FUNCTION_BLOCK "GCS7_LiftingDevice"	// FB 85
TITLE = MACHINE: Lifting Device
//  
//COPYRIGHT:    (C) 1997  BUHLER AG, CH-9240 UZWIL,  SWITZERLAND
//
//PRODUCT:      GCS7
//
//TITLE:        FB 85 MACHINE: Lifting Device (de:Hubzug)
// 
//-------------------------------------------------------------------------
//
//IDENT:        AUTHOR:             DEPT:                       DATE:
//FB85.2.4      M.Wedler            AEB31                       28-Jul-2008
//              Software counter with functions hardware's counter
//FB85.2.3      U.Kemmesies         AEB31                       07-Dez-2007
//              No Counter-Card
//FB85.2.2      M.Wedler            AEB31                       05-Jan-2007
//              BankingLoadingScrew for kilning box, calibration,
//              load counter value after failure, InEnableLowerMinPos
//FB85.2.1      M.Wedler            AEB31                       12-Sep-2006
//              Don't initialisation way counter by loading counter value
//FB85.2.0      A.Egli              CT3                         22-Mar-2006
//              ParPulseOnTime,ParPulseOffTime
//FB85.1.0      A.Egli              CT3                         22-Mar-2006
//              1st Release in S7
//
//-------------------------------------------------------------------------
//
//PURPOSE:      MANUAL : see [LL.xxMAN]
//
//RESTRICTIONS: S7
//
//-------------------------------------------------------------------------
//
AUTHOR : EA
FAMILY : GCS7LL
NAME : Lifting
VERSION : 2.3
VAR
  Ma : UDT 20850;
  MotorLeft : FB 12;	//Element Motor
  MotorRight : FB 12;	//Element Motor
  LSTopLeft : FB 14;	//LS top left side
  LSTopRight : FB 14;	//LS top right side
  LSTopStopLeft : FB 14;	//Emergency stop stop left
  LSTopStopRight : FB 14;	//Emergency stop stop right
  SMLeft : FB 14;	//Speed monitoring left side
  SMRight : FB 14;	//Speed monitoring right side
  OffTrackMon : FB 14;	//Track monitoring
  CounterLeft : UDT 20851;
  CounterRight : UDT 20851;
END_VAR
VAR_TEMP
  tmpFaultSum : BOOL ;
  tmpEnable : BOOL ;
  tmpLocal : BOOL ;
  tmpLenDyn : INT ;
  tmpOK : BOOL ;
  tmpDiff : INT ;
  tmpAddrIOLeft : DINT ;
  tmpAddrIORight : DINT ;
  tmpAddrCounterLeft : DINT ;
  tmpAddrCounterRight : DINT ;
  tmpAddrOffset : DINT ;
  tmpUnloadingActive : BOOL ;
END_VAR
BEGIN
NETWORK
TITLE =
      L     90;
      T     #tmpLenDyn;
NETWORK
TITLE = PC Control
//=== Test Object number =====================
      L     "SYS_DirectCtrlDB".PC.ObjectNo;	//PCControl.ObjectNo
      L     #Ma.Par.ParObjectNo;	//Input ObjectNo
      <>I;
      JC    aEnd;
//=== Test OType      ========================
      L     2085;	//Input object type
      L     "SYS_DirectCtrlDB".PC.ObjectType;	//PCControl.ObjectType
      <>I;
      JC    aEnd;
//=== Test Handshake =========================
      A     "SYS_DirectCtrlDB".PC.Hsk.FExamine;	// Handshake.FExamine
      JC    aExa;
      A     "SYS_DirectCtrlDB".PC.Hsk.FDefineCmd;	// Handshake.FDefineCmd
      O     "SYS_DirectCtrlDB".PC.Hsk.FDefinePara;	// Handshake.FDefinePara
      JC    aCmd;
      JU    aEnd;
// Write new commands from PC to Interface of group 
aCmd: A     "SYS_DirectCtrlDB".PC.Cmd1[8];	//Cmd1[8]=CmdOff
      S     #Ma.CmdOff;
      A     "SYS_DirectCtrlDB".PC.Cmd1[9];	//Cmd1[9]=CmdUp
      S     #Ma.CmdUp;
      A     "SYS_DirectCtrlDB".PC.Cmd1[10];	//Cmd1[10]=CmdNext
      S     #Ma.CmdNext;
      A     "SYS_DirectCtrlDB".PC.Cmd1[11];	//Cmd1[11]=CmdFaultReset
      S     #Ma.CmdFaultReset;
      A     "SYS_DirectCtrlDB".PC.Cmd1[13];	//Cmd1[13]=CmdManualOn
      S     #Ma.InManual;
      A     "SYS_DirectCtrlDB".PC.Cmd1[7];	//Cmd1[6]=CmdDown
      S     #Ma.CmdDown;
      A     "SYS_DirectCtrlDB".PC.Cmd2[13];	//Cmd2[13]=CmdManualOff
      R     #Ma.InManual;
//-----------------------------------------------------------
//Audit Log
aExa: NOP   0;
//------------------------------------------
      TAR2;	// Address Dynamic datas
      T     "SYS_DirectCtrlDB".GC.InDynAddr;	// -->PCControl.GC.InDynAddr
      L     #tmpLenDyn;	// Length Dynamic data
      T     "SYS_DirectCtrlDB".GC.InDynLen;	// -->PCControl.GC.InDynLen
      L     0;
      T     "SYS_DirectCtrlDB".GC.InParaAddr;	// -->PCControl.GC.InParaAddr
      T     "SYS_DirectCtrlDB".GC.InParaLen;	// -->PCControl.GC.InParaLen
      L     1;	// Code FcExamine
      UC    "SYS_DirectCtrl";
      L     10;	//Revision
      T     "SYS_DirectCtrlDB".GC.Revision;
aEnd: NOP   0;
NETWORK
TITLE = Calculate Address for Counter
      NOP   0;
//Calculate address for counter
      TAR2;
      L     DW#16#FFFFFF;
      AD;
      T     #tmpAddrOffset;
      L     P##CounterLeft;
      +D;
      T     #tmpAddrCounterLeft;
      L     #Ma.Par.ParIOByteNoCounterLeft;
      SLD   3;
      T     #tmpAddrIOLeft;
      L     #tmpAddrOffset;
      L     P##CounterRight;
      +D;
      T     #tmpAddrCounterRight;
      L     #Ma.Par.ParIOByteNoCounterRight;
      SLD   3;
      T     #tmpAddrIORight;
NETWORK
TITLE = Commands for Counter
//      L     0                           // [2.3]
//      L     #tmpAddrIOLeft              // [2.3]
//      ==D                               // [2.3]
////[2.4]     SPB   CTX0                        // [2.3]
//      SPB   IUK1                        // [2.4]
//      SPA   IUK0                        // [2.4]
//IUK1: NOP   0                           // [2.4]
////Calibration Zero                      // [2.4]
//      U     #Ma.InCalibration           // [2.4]
//      U     #Ma.InCalibrationZero       // [2.4]
//      U     #Ma.InPowerOk               // [2.4]
//      U     #Ma.InPowerOkDelayDone      // [2.4]
//      SPBN  IUK2                        // [2.4]
//      L     L#0                         // [2.4]
//      T     #CounterLeft.OutpSetCount   // [2.4]
//      T     #CounterRight.OutpSetCount  // [2.4]
//      T     #CounterLeft.VarInpHold     // [2.4]
//      T     #CounterRight.VarInpHold    // [2.4]
//      SET                               // [2.4]
//      S     #CounterLeft.OutpLOAD_VAL   // [2.4]
//      S     #CounterRight.OutpLOAD_VAL  // [2.4]
//IUK2: NOP   0                           // [2.4]
//      U     #CounterLeft.InpSTS_LOAD    // [2.4]
//      R     #CounterLeft.OutpLOAD_VAL   // [2.4]
//      U     #CounterRight.InpSTS_LOAD   // [2.4]
//      R     #CounterRight.OutpLOAD_VAL  // [2.4]
//      SPA   CTX0                        // [2.4]
//IUK0: NOP   0
      L     0;	// [2.3]
      L     #tmpAddrIOLeft;	// [2.3]
      ==D;	// [2.3]
//[2.4]     SPB   CTX0                        // [2.3]
      JC    IUK1;	// [2.4]
      JU    IUK0;	// [2.4]
IUK1: NOP   0;	// [2.4]
//Calibration Zero                      // [2.4]
      A     #Ma.InCalibration;	// [2.4]
      A     #Ma.InCalibrationZero;	// [2.4]
      A     #Ma.InPowerOk;	// [2.4]
      A     #Ma.InPowerOkDelayDone;	// [2.4]
      JCN   IUK2;	// [2.4]
      L     L#0;	// [2.4]
      T     #CounterLeft.InpActCount;	// [2.4]
      T     #CounterRight.InpActCount;	// [2.4]
      T     #CounterLeft.VarInpHold;	// [2.4]
      T     #CounterRight.VarInpHold;	// [2.4]
IUK2: NOP   0;	// [2.4]
      JU    CTX0;	// [2.4]
IUK0: NOP   0;
      NOP   0;
//Clear command or counter
      A     #Ma.InPowerOk;	// [2.2]
      A     #CounterLeft.OutpLOAD_VAL;	// [2.2]
      AN    #CounterLeft.InpSTS_LOAD;	// [2.2]
      JC    CTJ9;	// [2.2]
      LAR1  #tmpAddrCounterLeft;
      L     0;
      T     DID [AR1,P#4.0];
CTJ9: NOP   0;	// [2.2]
      A     #Ma.InPowerOk;	// [2.2]
      A     #CounterRight.OutpLOAD_VAL;	// [2.2]
      AN    #CounterRight.InpSTS_LOAD;	// [2.2]
      JC    CTJ8;	// [2.2]
      LAR1  #tmpAddrCounterRight;
      L     0;
      T     DID [AR1,P#4.0];
CTJ8: NOP   0;	// [2.2]
//---------------------------
      SET;
      S     #CounterLeft.OutpSW_GATE;
      S     #CounterRight.OutpSW_GATE;
//---------------------------
//Load counter value after failure      // [2.2]
      A     #Ma.InPowerOk;
      AN    #Ma.InPowerOkDelayDone;
      O;	// [2.2]
      A     #CounterLeft.OutpLOAD_VAL;	// [2.2]
      AN    #CounterLeft.InpSTS_LOAD;	// [2.2]
      JCN   CTJ2;	// [2.2]
      L     #CounterLeft.VarInpHold;
      T     #CounterLeft.OutpSetCount;
//    SET                               // [2.2]
      L     #CounterLeft.VarInpHold;	// [2.2]
      L     #CounterLeft.InpActCount;	// [2.2]
      <>D;	// [2.2]
      S     #CounterLeft.OutpLOAD_VAL;
CTJ2: NOP   0;	// [2.2]
      A     #Ma.InPowerOk;
      AN    #Ma.InPowerOkDelayDone;
      O;	// [2.2]
      A     #CounterRight.OutpLOAD_VAL;	// [2.2]
      AN    #CounterRight.InpSTS_LOAD;	// [2.2]
      JCN   CTJ1;
      L     #CounterRight.VarInpHold;
      T     #CounterRight.OutpSetCount;
//    SET                               // [2.2]
      L     #CounterRight.VarInpHold;	// [2.2]
      L     #CounterRight.InpActCount;	// [2.2]
      <>D;	// [2.2]
      S     #CounterRight.OutpLOAD_VAL;
CTJ1: NOP   0;
      A     #Ma.InPowerOk;
      A     #Ma.InPowerOkDelayDone;
      AN    #CounterLeft.InpSTS_LOAD;	// [2.2]
      AN    #CounterRight.InpSTS_LOAD;	// [2.2]
      AN    #CounterLeft.OutpLOAD_VAL;	// [2.2]
      AN    #CounterRight.OutpLOAD_VAL;	// [2.2]
      JCN   CTJ0;
      L     #CounterLeft.InpActCount;
      T     #CounterLeft.VarInpHold;
      L     #CounterRight.InpActCount;
      T     #CounterRight.VarInpHold;
CTJ0: NOP   0;
//Calibration Zero                      // [2.2]
      A     #Ma.InCalibration;	// [2.2]
      A     #Ma.InCalibrationZero;	// [2.2]
      A     #Ma.InPowerOk;	// [2.2]
      A     #Ma.InPowerOkDelayDone;	// [2.2]
      JCN   CTZ0;	// [2.2]
      L     L#0;	// [2.2]
      T     #CounterLeft.OutpSetCount;	// [2.2]
      T     #CounterRight.OutpSetCount;	// [2.2]
      T     #CounterLeft.VarInpHold;	// [2.2]
      T     #CounterRight.VarInpHold;	// [2.2]
      SET;	// [2.2]
      S     #CounterLeft.OutpLOAD_VAL;	// [2.2]
      S     #CounterRight.OutpLOAD_VAL;	// [2.2]
CTZ0: NOP   0;	// [2.2]
      A     #CounterLeft.InpSTS_LOAD;	// [2.2]
      R     #CounterLeft.OutpLOAD_VAL;	// [2.2]
      A     #CounterRight.InpSTS_LOAD;	// [2.2]
      R     #CounterRight.OutpLOAD_VAL;	// [2.2]
CTX0: NOP   0;	// [2.3]
NETWORK
TITLE = Initialisation way counter when in upper finally position 
//      L     0                           // [2.3]
//      L     #tmpAddrIOLeft              // [2.3]
//      ==D                               // [2.3]
////[2.4]      SPB   M050                        // [2.3]
//      SPB   UKI1                        // [2.4]
//      SPA   UKI0                        // [2.4]
//UKI1: NOP   0                           // [2.4]
//      UN    #Ma.InPowerOkDelayDone      // [2.4]
//      O     #Ma.InCalibration           // [2.4]
//      SPB   UKI2                        // [2.4]
//// Initialisation counter left when in end position top
//      O     #MotorLeft.StStartedFwd
//      O     #MotorLeft.StStopping
//      U     #LSTopLeft.StTrue
//      SPBN  UKI2
//      L     #Ma.Par.ParPositionTopLeftInc
//      ITD   
//      T     #CounterLeft.OutpSetCount
//      T     #CounterLeft.VarInpHold     // [2.4]
//      SET                               // [2.4]
//      S     #CounterLeft.OutpLOAD_VAL   // [2.4]
//UKI2: NOP   0
//      UN    #Ma.InPowerOkDelayDone      // [2.4]
//      O     #Ma.InCalibration           // [2.4]
//      SPB   UKI3                        // [2.4]
//// Initialisation counter rigth  when in end position top
//      O     #MotorRight.StStartedFwd
//      O     #MotorRight.StStopping
//      U     #LSTopRight.StTrue          // Endschalter oben
//      SPBN  UKI3
//      L     #Ma.Par.ParPositionTopRightInc
//      ITD   
//      T     #CounterRight.OutpSetCount
//      T     #CounterRight.VarInpHold    // [2.4]
//      SET                               // [2.4]
//      S     #CounterRight.OutpLOAD_VAL  // [2.4]
//UKI3: NOP   0                           // [2.4]
//      U     #CounterLeft.InpSTS_LOAD    // [2.4]
//      R     #CounterLeft.OutpLOAD_VAL   // [2.4]
//      U     #CounterRight.InpSTS_LOAD   // [2.4]
//      R     #CounterRight.OutpLOAD_VAL  // [2.4]
//      SPA   M050                        // [2.4]
//UKI0: NOP   0                           // [2.4]
//
      L     0;	// [2.3]
      L     #tmpAddrIOLeft;	// [2.3]
      ==D;	// [2.3]
//[2.4]      SPB   M050                        // [2.3]
      JC    UKI1;	// [2.4]
      JU    UKI0;	// [2.4]
UKI1: NOP   0;	// [2.4]
      AN    #Ma.InPowerOkDelayDone;	// [2.4]
      O     #Ma.InCalibration;	// [2.4]
      JC    UKI2;	// [2.4]
// Initialisation counter left when in end position top
      O     #MotorLeft.StStartedFwd;
      O     #MotorLeft.StStopping;
      A     #LSTopLeft.StTrue;
      JCN   UKI2;
      L     #Ma.Par.ParPositionTopLeftInc;
      ITD;
      T     #CounterLeft.InpActCount;	// [2.4]
      T     #CounterLeft.VarInpHold;	// [2.4]
UKI2: NOP   0;
      AN    #Ma.InPowerOkDelayDone;	// [2.4]
      O     #Ma.InCalibration;	// [2.4]
      JC    UKI3;	// [2.4]
// Initialisation counter rigth  when in end position top
      O     #MotorRight.StStartedFwd;
      O     #MotorRight.StStopping;
      A     #LSTopRight.StTrue;	// Endschalter oben
      JCN   UKI3;
      L     #Ma.Par.ParPositionTopRightInc;
      ITD;
      T     #CounterRight.InpActCount;	// [2.4]
      T     #CounterRight.VarInpHold;	// [2.4]
UKI3: NOP   0;	// [2.4]
      JU    M050;	// [2.4]
UKI0: NOP   0;	// [2.4]
      NOP   0;
//-------------------------------------------------------
      A     #CounterLeft.InpSTS_LOAD;	// [2.1]
      ON    #Ma.InPowerOkDelayDone;	// [2.1]
      O     #Ma.InCalibration;	// [2.2]
      JC    M051;	// [2.1]
// Initialisation counter left when in end position top
      O     #MotorLeft.StStartedFwd;
      O     #MotorLeft.StStopping;
      A     #LSTopLeft.StTrue;
      JCN   M051;
      L     #Ma.Par.ParPositionTopLeftInc;
      ITD;
      T     #CounterLeft.OutpSetCount;
      T     #CounterLeft.VarInpHold;	// [2.2]
//Set Write command 
      L     #Ma.Par.ParPositionTopLeftInc;
      L     #Ma.OutIncrementLeft;
      <>I;
      S     #CounterLeft.OutpLOAD_VAL;	//--> Command to counter to set target value
M051: NOP   0;
//-------------------------------------------------------
      A     #CounterRight.InpSTS_LOAD;	// [2.1]
      ON    #Ma.InPowerOkDelayDone;	// [2.1]
      O     #Ma.InCalibration;	// [2.2]
      JC    M052;	// [2.1]
// Initialisation counter rigth  when in end position top
      O     #MotorRight.StStartedFwd;
      O     #MotorRight.StStopping;
      A     #LSTopRight.StTrue;	// Endschalter oben
      JCN   M052;
      L     #Ma.Par.ParPositionTopRightInc;
      ITD;
      T     #CounterRight.OutpSetCount;
      T     #CounterRight.VarInpHold;	// [2.2]
//Set Write command
      L     #Ma.Par.ParPositionTopRightInc;
      L     #Ma.OutIncrementRight;
      <>I;
      S     #CounterRight.OutpLOAD_VAL;	//--> Command to counter to set target value
M052: NOP   0;
M050: NOP   0;	// [2.3]
NETWORK
TITLE = Read Global Command
      A     "GCS7_Gr_OutFaultReset";	// OutFaultReset
      S     #Ma.CmdFaultReset;
NETWORK
TITLE = Write Outputs of counter
      L     0;
      L     #tmpAddrIOLeft;
      ==D;
      JC    WCJ0;
//Write Outputs  Counter left
      LAR1  #tmpAddrCounterLeft;
      L     DID [AR1,P#0.0];
      LAR1  #tmpAddrIOLeft;
      T     PQD [AR1,P#0.0];
      LAR1  #tmpAddrCounterLeft;
      L     DID [AR1,P#4.0];
      LAR1  #tmpAddrIOLeft;
      T     PQD [AR1,P#4.0];
//Write Outputs Counter right
      LAR1  #tmpAddrCounterRight;
      L     DID [AR1,P#0.0];
      LAR1  #tmpAddrIORight;
      T     PQD [AR1,P#0.0];
      LAR1  #tmpAddrCounterRight;
      L     DID [AR1,P#4.0];
      LAR1  #tmpAddrIORight;
      T     PQD [AR1,P#4.0];
WCJ0: NOP   0;
NETWORK
TITLE = Read Counter
      L     0;
      L     #tmpAddrIOLeft;
      ==D;
      JC    WRJ0;
//Read IO Counter left
      LAR1  #tmpAddrIOLeft;
      L     PID [AR1,P#0.0];
      LAR1  #tmpAddrCounterLeft;
      T     DID [AR1,P#8.0];
      LAR1  #tmpAddrIOLeft;
      L     PID [AR1,P#4.0];
      LAR1  #tmpAddrCounterLeft;
      T     DID [AR1,P#12.0];
//Read IO Counter right
      LAR1  #tmpAddrIORight;
      L     PID [AR1,P#0.0];
      LAR1  #tmpAddrCounterRight;
      T     DID [AR1,P#8.0];
      LAR1  #tmpAddrIORight;
      L     PID [AR1,P#4.0];
      LAR1  #tmpAddrCounterRight;
      T     DID [AR1,P#12.0];
WRJ0: NOP   0;
NETWORK
TITLE = Calculate: mm per incement 
      L     #Ma.Par.ParPositionTopLeftUnits;
      DTR;
      L     #Ma.Par.ParPositionTopLeftInc;	//Hoehe Endschalter 
      DTR;
      /R;
      T     #Ma.Par.OutUnitsPerIncLeft;
      L     #Ma.Par.ParPositionTopRightUnits;
      DTR;
      L     #Ma.Par.ParPositionTopRightInc;	//Hoehe Endschalter 
      DTR;
      /R;
      T     #Ma.Par.OutUnitsPerIncRight;
NETWORK
TITLE = Speed Monitoring Lifting 
      NOP   0;
//==========================================================
//Speed Monitoring Left
//==========================================================
//- Check if increment is changing
      A(;
      L     #CounterLeft.InpActCount;
      L     #Ma.OutIncrementLeft;
      ==D;
      );
      A(;
      O     #MotorLeft.OutpRunFwd;
      O     #MotorLeft.OutpRunRev;
      );
      AN    #Ma.CmdFaultReset;
      JC    M1J1;
      L     #Ma.Par.ParMonTime;	//5s
      T     #Ma.Par.OutMonTimeLeft;
      S     #SMLeft.InpTrue;
//---Run monitoring time
M1J1: AN    "GCS7_Gr_OutTick200ms";
      JC    M1J2;
      L     #Ma.Par.OutMonTimeLeft;
      +     -2;
      T     #Ma.Par.OutMonTimeLeft;
      L     0;
      >=I;
      JC    M1J2;
      T     #Ma.Par.OutMonTimeLeft;
      R     #SMLeft.InpTrue;
//---Store old counter value
M1J2: L     #CounterLeft.InpActCount;
      T     #Ma.OutIncrementLeft;
//==========================================================
//Speed Monitoring Right
//==========================================================
//- Check if increment is changing
      A(;
      L     #CounterRight.InpActCount;
      L     #Ma.OutIncrementRight;
      ==D;
      );
      A(;
      O     #MotorRight.OutpRunFwd;
      O     #MotorRight.OutpRunRev;
      );
      AN    #Ma.CmdFaultReset;
      JC    M2J1;
      L     #Ma.Par.ParMonTime;	//5s
      T     #Ma.Par.OutMonTimeRight;
      S     #SMRight.InpTrue;
//---Run monitoring time
M2J1: AN    "GCS7_Gr_OutTick200ms";
      JC    M2J2;
      L     #Ma.Par.OutMonTimeRight;
      +     -2;
      T     #Ma.Par.OutMonTimeRight;
      L     0;
      >=I;
      JC    M2J2;
      T     #Ma.Par.OutMonTimeRight;
      R     #SMRight.InpTrue;
//---Store old counter value
M2J2: L     #CounterRight.InpActCount;
      T     #Ma.OutIncrementRight;
NETWORK
TITLE = Calculation position in mm
// Zaehlwert Hubzug 1 in mm umrechnen
      L     #Ma.OutIncrementLeft;
      DTR;
      L     #Ma.Par.OutUnitsPerIncLeft;
      *R;
      RND;
      T     #Ma.OutPositionLeft;
// Zaehlwert Hubzug 2 in mm umrechnen
      L     #Ma.OutIncrementRight;
      DTR;
      L     #Ma.Par.OutUnitsPerIncRight;
      *R;
      RND;
      T     #Ma.OutPositionRight;
NETWORK
TITLE = Check maximum difference position to stop 1 motor 
      NOP   0;
//---Check Position left to high
      L     #Ma.OutPositionLeft;
      L     #Ma.BankingLoadingScrew;	// [2.2]
      +I;	// [2.2]
      L     #Ma.OutPositionRight;
      -I;
      T     #Ma.OutPositionDifference;
      L     #Ma.Par.ParMaxOffTrackPause;
      >=I;
      S     #Ma.OutPositionLeftToHigh;
      L     #Ma.OutPositionRight;
      L     #Ma.BankingLoadingScrew;	// [2.2]
      -I;	// [2.2]
      L     #Ma.OutPositionLeft;
      >=I;
      R     #Ma.OutPositionLeftToHigh;
//---Check position right to high
      L     #Ma.OutPositionRight;
      L     #Ma.BankingLoadingScrew;	// [2.2]
      -I;	// [2.2]
      L     #Ma.OutPositionLeft;
      -I;
      L     #Ma.Par.ParMaxOffTrackPause;
      >=I;
      S     #Ma.OutPositionRightToHigh;
      L     #Ma.OutPositionRight;
      L     #Ma.BankingLoadingScrew;	// [2.2]
      -I;	// [2.2]
      L     #Ma.OutPositionLeft;
      <=I;
      R     #Ma.OutPositionRightToHigh;
NETWORK
TITLE = Check maximum difference position to generate fault
      L     #Ma.OutPositionLeft;
      L     #Ma.OutPositionRight;
      -I;
      JP    DIJ1;
      NEGI;
DIJ1: L     #Ma.Par.ParMaxOffTrackFault;
      >=I;
      =     #Ma.OutDifferenceFault;
NETWORK
TITLE = Check Minimum position
      A(;
      L     #Ma.OutPositionLeft;
      L     #Ma.Par.ParPositionMin;
      >=I;
      );
      A(;
      L     #Ma.OutPositionRight;
      L     #Ma.Par.ParPositionMin;
      >=I;
      );
      =     #Ma.OutHigherMinPos;
NETWORK
TITLE = Check Adjusted
      NOP   0;
//------------------
      L     #Ma.OutPositionLeft;
      L     #Ma.InPositionTarget;
      -I;
      JP    A1J1;
      NEGI;
A1J1: L     #Ma.Par.ParTolPosition;
      <=I;
      =     #Ma.OutAdjustedLeft;
//------------------
      L     #Ma.OutPositionRight;
      L     #Ma.BankingLoadingScrew;	// [2.2]
      -I;	// [2.2]
      L     #Ma.InPositionTarget;
      -I;
      JP    A2J1;
      INVI;
A2J1: L     #Ma.Par.ParTolPosition;
      <=I;
      =     #Ma.OutAdjustedRight;
//------------------
NETWORK
TITLE = Interlocking
//===Global Group Orders===
      A     "GCS7_Gr_OutManualOff";	//Gr.OutManualOff
      R     #Ma.InManual;
      A     #Ma.InManual;
      S     "GCS7_Gr_InManual";	//Gr.InManual
//--------------
      A     #Ma.CmdUp;
      S     #Ma.OutManStartReqUp;
      R     #Ma.OutManStartReqDown;
      A     #Ma.CmdDown;
      R     #Ma.OutManStartReqUp;
      S     #Ma.OutManStartReqDown;
      A     #Ma.CmdOff;
      ON    #Ma.InManual;
      R     #Ma.OutManStartReqUp;
      R     #Ma.OutManStartReqDown;
//--- Fault----
      A     #MotorLeft.StFault;
      O     #MotorRight.StFault;
      O     #LSTopLeft.StFault;
      O     #LSTopRight.StFault;
      O     #LSTopStopLeft.StFault;
      O     #LSTopStopRight.StFault;
      O     #SMLeft.StFault;
      O     #SMRight.StFault;
      O     #OffTrackMon.StFault;
      =     #tmpFaultSum;
//--- InLocal----
      A     #Ma.InLocal;
      AN    #Ma.InManual;
      =     #tmpLocal;
      =     #MotorLeft.InLocal;
      =     #MotorRight.InLocal;
      =     #LSTopLeft.InLocal;
      =     #LSTopRight.InLocal;
      =     #LSTopStopLeft.InLocal;
      =     #LSTopStopRight.InLocal;
      =     #SMLeft.InLocal;
      =     #SMRight.InLocal;
      =     #OffTrackMon.InLocal;
//--- Fault Reset -------------
      A     #Ma.CmdFaultReset;
      S     #MotorLeft.CmdFaultReset;
      S     #MotorRight.CmdFaultReset;
      S     #LSTopLeft.CmdFaultReset;
      S     #LSTopRight.CmdFaultReset;
      S     #LSTopStopLeft.CmdFaultReset;
      S     #LSTopStopRight.CmdFaultReset;
      S     #SMLeft.CmdFaultReset;
      S     #SMRight.CmdFaultReset;
      S     #OffTrackMon.CmdFaultReset;
NETWORK
TITLE = Start as Pulse during unloading [2.0]
      A     #Ma.InEnableUp;	//[2.0]
      O     #Ma.InEnableDown;	//[2.0]
      AN    #tmpLocal;	//[2.0]
      AN    #Ma.InManual;	//[2.0]
      AN    #Ma.CmdOff;	//[2.0]
      AN    #Ma.StAdjusted;	//[2.0]
      AN    #tmpFaultSum;	//[2.0]
      A     #Ma.InUnloading;	//[2.0]
      =     #tmpUnloadingActive;	//[2.0]
      AN    #tmpUnloadingActive;	//[2.0]
      R     #Ma.OutPulseOn;	//[2.0]
      L     0;	//[2.0]
      JC    PuJ3;	//[2.0]
//--Decrement pulse time --
      AN    "GCS7_Gr_OutTick200ms";	//[2.0]
      L     #Ma.OutPulseTime;	//[2.0]
      JC    PuJ4;	//[2.0]
      +     -2;	//[2.0]
      T     #Ma.OutPulseTime;	//[2.0]
PuJ4: L     0;	//[2.0]
      >I;	//[2.0]
      JC    PuJ1;	//[2.0]
      AN    #Ma.OutPulseOn;	//[2.0]
      S     #Ma.OutPulseOn;	//[2.0]
      L     #Ma.Par.ParPulseOffTime;	//[2.0]
      JC    PuJ3;	//[2.0]
      R     #Ma.OutPulseOn;	//[2.0]
      L     #Ma.Par.ParPulseOnTime;	//[2.0]
PuJ3: T     #Ma.OutPulseTime;	//[2.0]
PuJ1: NOP   0;	//[2.0]
NETWORK
TITLE = Interlocking Motor Left
      L     #Ma.OutIncrementLeft;
      L     0;
      >I;
      AN    #tmpFaultSum;
      ON    #Ma.InInterlocked;
      A     #Ma.InEnableDown;
      A(;
      L     #Ma.InPositionTarget;
      L     #Ma.OutPositionLeft;
      <I;
      AN    #Ma.OutAdjustedLeft;
      AN    #Ma.InManual;
      A(;
      ON    #Ma.InUnloading;	//[2.0]
      ON    #Ma.OutPulseOn;	//[2.0]
      );
      O     #Ma.OutManStartReqDown;
      );
      AN    #Ma.OutPositionRightToHigh;
      AN    #Ma.OutDifferenceFault;
      A     #Ma.InEnableDown;
      A     #Ma.InEnableLowerMinPos;	//[2.2]
      A     #Ma.InPowerOkDelayDone;
      =     #MotorLeft.InEnableRev;
      AN    #tmpFaultSum;
      A     #LSTopLeft.StFalse;
      A     #LSTopStopLeft.StFalse;
      ON    #Ma.InInterlocked;
      A     #Ma.InEnableDown;
      A(;
      L     #Ma.InPositionTarget;
      L     #Ma.OutPositionLeft;
      >I;
      AN    #Ma.OutAdjustedLeft;
      AN    #Ma.InManual;
      A(;
      ON    #Ma.InUnloading;	//[2.0]
      ON    #Ma.OutPulseOn;	//[2.0]
      );
      O     #Ma.OutManStartReqUp;
      );
      AN    #Ma.OutPositionLeftToHigh;
      A     #Ma.InEnableUp;
      AN    #Ma.OutDifferenceFault;
      A     #Ma.InPowerOkDelayDone;
      =     #MotorLeft.InEnableFwd;
      A     #Ma.CmdNext;
      O     #Ma.InManual;
      S     #MotorLeft.CmdNext;
NETWORK
TITLE = Interlocking Motor Right
      L     #Ma.OutIncrementRight;
      L     0;
      >I;
      AN    #tmpFaultSum;
      ON    #Ma.InInterlocked;
      A     #Ma.InEnableDown;
      A(;
      L     #Ma.InPositionTarget;
      L     #Ma.BankingLoadingScrew;	//[2.2]
      +I;	//[2.2]
      L     #Ma.OutPositionRight;
      <I;
      AN    #Ma.OutAdjustedRight;
      AN    #Ma.InManual;
      A(;
      ON    #Ma.InUnloading;	//[2.0]
      ON    #Ma.OutPulseOn;	//[2.0]
      );
      O     #Ma.OutManStartReqDown;
      );
      AN    #Ma.OutPositionLeftToHigh;
      AN    #Ma.OutDifferenceFault;
      A     #Ma.InEnableDown;
      A     #Ma.InEnableLowerMinPos;	//[2.2]
      A     #Ma.InPowerOkDelayDone;
      =     #MotorRight.InEnableRev;
      AN    #tmpFaultSum;
      A     #LSTopRight.StFalse;
      A     #LSTopStopRight.StFalse;
      ON    #Ma.InInterlocked;
      A     #Ma.InEnableDown;
      A(;
      L     #Ma.InPositionTarget;
      L     #Ma.BankingLoadingScrew;	//[2.2]
      +I;	//[2.2]
      L     #Ma.OutPositionRight;
      >I;
      AN    #Ma.OutAdjustedRight;
      AN    #Ma.InManual;
      A(;
      ON    #Ma.InUnloading;	//[2.0]
      ON    #Ma.OutPulseOn;	//[2.0]
      );
      O     #Ma.OutManStartReqUp;
      );
      AN    #Ma.OutPositionRightToHigh;
      AN    #Ma.OutDifferenceFault;
      A     #Ma.InEnableUp;
      A     #Ma.InPowerOkDelayDone;
      =     #MotorRight.InEnableFwd;
      A     #Ma.CmdNext;
      O     #Ma.InManual;
      S     #MotorRight.CmdNext;
NETWORK
TITLE = Interlocking LSTopStopLeft, LSTopStopRight,LSTopLeft,LSTopRigh
//Mointoring false
//When started downwards, the the LS must be uncovered after 30 mm
//
//
      CLR;
      =     #LSTopStopLeft.InMonTrue;
      =     #LSTopStopRight.InMonTrue;
      CLR;
      =     #LSTopLeft.InMonTrue;
      =     #LSTopRight.InMonTrue;
//Monitoring false
      L     #Ma.Par.ParPositionTopLeftUnits;
      L     #Ma.OutPositionLeft;
      -I;
      L     30;	//30mms
      >=I;
      A     #MotorLeft.StStartedRev;
      A     #Ma.InInterlocked;
      =     #LSTopLeft.InMonFalse;
      SET;
      =     #LSTopStopLeft.InMonFalse;
      L     #Ma.Par.ParPositionTopRightUnits;
      L     #Ma.OutPositionRight;
      -I;
      L     30;	//30mms
      >=I;
      A     #MotorRight.StStartedRev;
      A     #Ma.InInterlocked;
      =     #LSTopRight.InMonFalse;
      SET;
      =     #LSTopStopRight.InMonFalse;
NETWORK
TITLE = Control Element SMLeft, SMRight
      A     #MotorLeft.StStartedRev;
      O     #MotorLeft.StStartedFwd;
      =     #SMLeft.InMonTrue;
      A     #MotorRight.StStartedRev;
      O     #MotorRight.StStartedFwd;
      =     #SMRight.InMonTrue;
NETWORK
TITLE = Control Element OffTrackMon
      AN    #Ma.OutDifferenceFault;
      =     #OffTrackMon.InpTrue;
      SET;
      =     #OffTrackMon.InMonTrue;
NETWORK
TITLE = Call Motor Left
      CALL  #MotorLeft;
NETWORK
TITLE = Call Motor Right
      CALL  #MotorRight;
NETWORK
TITLE = Call Digital Input: LSTopLeft
      CALL  #LSTopLeft;
NETWORK
TITLE = Call Digital Input: LSTopRight
      CALL  #LSTopRight;
NETWORK
TITLE = Call Digital Input: LSStopLeft
      CALL  #LSTopStopLeft;
NETWORK
TITLE = Call Digital Input: LSStopRight
      CALL  #LSTopStopRight;
NETWORK
TITLE = Call Digital Input: SMLeft
      CALL  #SMLeft;
NETWORK
TITLE = Call Digital Input: SMRight
      CALL  #SMRight;
NETWORK
TITLE = Call Digital Input: OffTrackMon
      CALL  #OffTrackMon;
NETWORK
TITLE = States
      A     #Ma.StStopped;
      JC    S0;
      A     #Ma.StAdjusted;
      JC    S6;
      A     #Ma.StStartedUP;
      JC    S2;
      A     #Ma.StStartedDown;
      JC    S5;
      A     #Ma.StStopping;
      JC    S3;
      A     #Ma.StStarting;
      JC    S1;
      A     #Ma.StFault;
      JC    S4;
      JU    xxS0;	//Initialise: goto StStopped
NETWORK
TITLE = StStopped
xxS0: S     #Ma.StStopped;
      JU    SAVE;
//---Transition -> StFault
S0:   A     #tmpFaultSum;
      R     #Ma.StStopped;
      JC    xxS4;
//---Transition -> StStarting
      A     #Ma.OutManStartReqDown;
      O     #Ma.OutManStartReqUp;
      A     #Ma.InManual;
      ON    #MotorLeft.StStopped;
      ON    #MotorRight.StStopped;
      R     #Ma.StStopped;
      JC    xxS1;
//---Transition for StAdjusted
      A     #Ma.OutAdjustedLeft;
      A     #Ma.OutAdjustedRight;
      AN    #tmpLocal;
      R     #Ma.StStopped;
      JC    xxS6;
      JU    SAVE;
NETWORK
TITLE = StStarting
//== Any transition to StStarting
xxS1: SET;
      S     #Ma.StStarting;
      JU    SAVE;
//== Logic ====
//---Transition -> StFault
S1:   A     #tmpFaultSum;
      R     #Ma.StStarting;
      JC    xxS4;
//---Transition -> StStartedUn
      A     #MotorLeft.StStartedFwd;
      O     #MotorRight.StStartedFwd;
      R     #Ma.StStarting;
      JC    xxS2;
//---Transition -> StStartingDown
      A     #MotorLeft.StStartedRev;
      O     #MotorRight.StStartedRev;
      R     #Ma.StStarting;
      JC    xxS5;
//---Transition for StStopping
      A     #MotorLeft.StStopped;
      A     #MotorRight.StStopped;
      AN    #Ma.OutManStartReqDown;
      AN    #Ma.OutManStartReqUp;
      O     #tmpLocal;
      R     #Ma.StStarting;
      JC    xxS3;
//---Transition for StAdjusted
      A     #Ma.OutAdjustedLeft;
      A     #Ma.OutAdjustedRight;
      AN    #tmpLocal;
      R     #Ma.StStarting;
      JC    xxS6;
      JU    SAVE;
NETWORK
TITLE = StStartedUp
xxS2: SET;
      S     #Ma.StStartedUP;
      JU    SAVE;
//---Transition -> StFault
S2:   A     #tmpFaultSum;	//---Condition for StFault
      R     #Ma.StStartedUP;
      JC    xxS4;
//---Transition for StAdjusted
      A     #Ma.OutAdjustedLeft;
      A     #Ma.OutAdjustedRight;
      R     #Ma.StStartedUP;
      JC    xxS3;
//---Transition -> StStoppting
      AN    #MotorLeft.StStartedFwd;
      AN    #MotorRight.StStartedFwd;
      AN    #tmpUnloadingActive;	//[2.0]
      O     #MotorLeft.StStartedRev;	//[2.0]
      O     #MotorRight.StStartedRev;	//[2.0]
      R     #Ma.StStartedUP;
      JC    xxS3;
      JU    SAVE;
NETWORK
TITLE = StStartedDown
xxS5: SET;
      S     #Ma.StStartedDown;
      JU    SAVE;
//---Transition -> StFault
S5:   A     #tmpFaultSum;	//---Condition for StFault
      R     #Ma.StStartedDown;
      JC    xxS4;
//---Transition for StAdjusted
      A     #Ma.OutAdjustedLeft;
      A     #Ma.OutAdjustedRight;
      R     #Ma.StStartedDown;
      JC    xxS3;
//---Transition -> StStoppting
      AN    #MotorLeft.StStartedRev;
      AN    #MotorRight.StStartedRev;
      AN    #tmpUnloadingActive;	//[2.0]
      O     #MotorLeft.StStartedFwd;	//[2.0]
      O     #MotorRight.StStartedFwd;	//[2.0]
      R     #Ma.StStartedDown;
      JC    xxS3;
      JU    SAVE;
NETWORK
TITLE = StAdjusted
xxS6: SET;
      S     #Ma.StAdjusted;
//---Transition -> StFault
S6:   A     #tmpFaultSum;
      R     #Ma.StAdjusted;
      JC    xxS4;
//---Transition for StStarting
      AN    #MotorLeft.StStopped;
      ON    #MotorRight.StStopped;
      R     #Ma.StAdjusted;
      JC    xxS1;
//---Transition -> StStopping
      AN    #Ma.OutAdjustedLeft;
      ON    #Ma.OutAdjustedRight;
      O     #tmpLocal;
      R     #Ma.StAdjusted;
      JC    xxS3;
      JU    SAVE;
NETWORK
TITLE = StStopping
//===Any transition to StStopping
xxS3: SET;
      S     #Ma.StStopping;
      JU    SAVE;
//===Logic =======================
//---Transtition -> StFault
S3:   A     #tmpFaultSum;
      R     #Ma.StStopping;
      JC    xxS4;
//---Transition -> StAdjusted
      A     #Ma.OutAdjustedLeft;
      A     #Ma.OutAdjustedRight;
      A     #MotorLeft.StStopped;
      A     #MotorRight.StStopped;
      AN    #tmpLocal;
      R     #Ma.StStopping;
      JC    xxS6;
//---Transition -> StStopped
      A     #MotorLeft.StStopped;
      A     #MotorRight.StStopped;
      R     #Ma.StStopping;
      JC    xxS0;
//---Transition -> StStarting
      AN    #MotorLeft.StStopping;
      AN    #MotorRight.StStopping;
      R     #Ma.StStopping;
      JC    xxS1;
      JU    SAVE;
NETWORK
TITLE =  StFault
// Any transiton to Fault  
xxS4: SET;
      S     #Ma.StFault;
//===logic
//---Transition -> StStopping
S4:   AN    #tmpFaultSum;
      R     #Ma.StFault;
      JC    xxS3;
      JU    SAVE;
NETWORK
TITLE = Global End
SAVE: SET;	//---Clear all commands
      R     #Ma.CmdUp;
      R     #Ma.CmdDown;
      R     #Ma.CmdOff;
      R     #Ma.CmdNext;
      R     #Ma.CmdFaultReset;
//---------------------------------
      AN    #MotorLeft.StStarting;
      AN    #MotorLeft.StStartedFwd;
      AN    #MotorLeft.StStartedRev;
      AN    #MotorRight.StStarting;
      AN    #MotorRight.StStartedFwd;
      AN    #MotorRight.StStartedRev;
      ON    #Ma.InManual;
      R     #Ma.OutManStartReqDown;
      R     #Ma.OutManStartReqUp;
NETWORK
TITLE = State Code
//--Stopped, Substate ---
      A     #Ma.StStopped;
      L     1;
      JC    STC9;
      A     #Ma.StStarting;
      L     2;
      JC    STC9;
      A     #Ma.StStartedUP;
      L     3;
      JC    STC9;
      A     #Ma.StStartedDown;
      L     5;
      JC    STC9;
      A     #Ma.StAdjusted;
      L     6;
      JC    STC9;
      A     #Ma.StStopping;
      L     7;
      JC    STC9;
      L     32;	// Code: fault
STC9: L     #Ma.StCode;	// Old state code
      TAK;
      T     #Ma.StCode;	// Save state code
      <>I;
      L     3;	// Load code for CBit methode
      CC    "SYS_CBitCtrl";
END_FUNCTION_BLOCK

FUNCTION_BLOCK "GCS7_TractionDrive"	// FB 86
TITLE = MACHINE: Traction Drive (de:Fahrantrieb)
//  
//COPYRIGHT:    (C) 1997  BUHLER AG, CH-9240 UZWIL,  SWITZERLAND
//
//PRODUCT:      GCS7
//
//TITLE:        FB 86 MACHINE: Traction Drive (de:Fahrantrieb)
// 
//-------------------------------------------------------------------------
//
//IDENT:        AUTHOR:             DEPT:                       DATE:
//FB86.1.11     M.Wedler            AEB41                       06-Nov-2008
//              Cleaning work after changes [1.8]                        
//FB86.1.10     M.Wedler            AEB41                       15-Okt-2008
//              Delay start motor by loading if flow detector is covered.
//FB86.1.9      M.Wedler            AEB41                       04-Feb-2008
//              No Counter-Card with Counter Rounds
//FB86.1.8      U.Kemmesies         AEB31                       07-Dez-2007
//              No Counter-Card
//FB86.1.7      M.Wedler            AEB31                       05-Jan-2007
//              Load counter value after failure
//FB86.1.6      U.Kemmesies         AEB31                       23-Nov-2006
//              Round counter only for Inkremental-Counter               
//FB86.1.5      U.Kemmesies         AEB31                       14-Nov-2006
//              Round counter               
//FB86.1.4      M.Wedler            AEB31                       12-Sep-2006
//              Don't reset "#Ma.CmdSetZeroPoint" after each cycle.               
//FB86.1.3      J.Voss              AEB31                       31-Aug-2006
//              Never clear setpoint speed [#Speed.InOutValuePc]
//FB86.1.2      M.Wedler            AEB31                       31-Aug-2006
//              Round counter forward and reverse for manual     
//              and automatic mode. Stop motor by loading if
//              flow detector is not covered.
//FB86.1.1      A.Egli              CT3                         31-Aug-2006
//              Count forward and reverse
//FB86.1.0      A.Egli              CT3                         22-Mar-2006
//              1st Release in S7
//
//-------------------------------------------------------------------------
//
//PURPOSE:      MANUAL : see [LL.xxMAN]
//
//RESTRICTIONS: S7
//
//-------------------------------------------------------------------------
//
AUTHOR : EA
FAMILY : GCS7LL
NAME : StrokeDr
VERSION : 1.8
VAR
  Ma : UDT 20860;
  Motor : FB 12;	//Element Motor
  Speed : FB 17;	//Element Analog output
  LSZeroPoint : FB 14;	//LS zero point
  Product : FB 14;	//Level probe
  SM : FB 14;	//Speed monitoring
  IncCounter : UDT 20851;
END_VAR
VAR_TEMP
  tmpFaultStop : BOOL ;
  tmpFaultSum : BOOL ;
  tmpEnable : BOOL ;
  tmpLocal : BOOL ;
  tmpLenDyn : INT ;
  tmpOK : BOOL ;
  tmpTestTime : INT ;
  tmpAddrIO : DINT ;
  tmpAddrCounter : DINT ;
  tmpAddrOffset : DINT ;
  tmpAdjusted : BOOL ;
  tmpStartPosition : BOOL ;
  tmpAngle1 : INT ;
  tmpAngleLes355 : BOOL ;
  tmpAngleDelta : INT ;
END_VAR
BEGIN
NETWORK
TITLE =
      L     80;
      T     #tmpLenDyn;
NETWORK
TITLE = PC Control
//=== Test Object number =====================
      L     "SYS_DirectCtrlDB".PC.ObjectNo;	//PCControl.ObjectNo
      L     #Ma.Par.ParObjectNo;	//Input ObjectNo
      <>I;
      JC    aEnd;
//=== Test OType      ========================
      L     2086;	//Input object type
      L     "SYS_DirectCtrlDB".PC.ObjectType;	//PCControl.ObjectType
      <>I;
      JC    aEnd;
//=== Test Handshake =========================
      A     "SYS_DirectCtrlDB".PC.Hsk.FExamine;	// Handshake.FExamine
      JC    aExa;
      A     "SYS_DirectCtrlDB".PC.Hsk.FDefineCmd;	// Handshake.FDefineCmd
      O     "SYS_DirectCtrlDB".PC.Hsk.FDefinePara;	// Handshake.FDefinePara
      JC    aCmd;
      JU    aEnd;
// Write new commands from PC to Interface of group 
aCmd: A     "SYS_DirectCtrlDB".PC.Cmd1[8];	//Cmd1[8]=CmdOff
      S     #Ma.CmdOff;
      A     "SYS_DirectCtrlDB".PC.Cmd1[9];	//Cmd1[9]=CmdUp
      S     #Ma.CmdOnFwd;
      A     "SYS_DirectCtrlDB".PC.Cmd1[10];	//Cmd1[10]=CmdNext
      S     #Ma.CmdNext;
      A     "SYS_DirectCtrlDB".PC.Cmd1[11];	//Cmd1[11]=CmdFaultReset
      S     #Ma.CmdFaultReset;
      A     "SYS_DirectCtrlDB".PC.Cmd1[13];	//Cmd1[13]=CmdManualOn
      S     #Ma.InManual;
      A     "SYS_DirectCtrlDB".PC.Cmd1[7];	//Cmd1[6]=CmdRev
      S     #Ma.CmdOnRev;
      A     "SYS_DirectCtrlDB".PC.Cmd2[13];	//Cmd2[13]=CmdManualOff
      R     #Ma.InManual;
//-----------------------------------------------------------
//Audit Log
aExa: NOP   0;
//------------------------------------------
      TAR2;	// Address Dynamic datas
      T     "SYS_DirectCtrlDB".GC.InDynAddr;	// -->PCControl.GC.InDynAddr
      L     #tmpLenDyn;	// Length Dynamic data
      T     "SYS_DirectCtrlDB".GC.InDynLen;	// -->PCControl.GC.InDynLen
      L     0;
      T     "SYS_DirectCtrlDB".GC.InParaAddr;	// -->PCControl.GC.InParaAddr
      T     "SYS_DirectCtrlDB".GC.InParaLen;	// -->PCControl.GC.InParaLen
      L     1;	// Code FcExamine
      UC    "SYS_DirectCtrl";
      L     10;	//Revision
      T     "SYS_DirectCtrlDB".GC.Revision;
aEnd: NOP   0;
NETWORK
TITLE = Calculate Address for Counter
      NOP   0;
//Calculate address for counter
      TAR2;
      L     DW#16#FFFFFF;
      AD;
      T     #tmpAddrOffset;
      L     P##IncCounter;
      +D;
      T     #tmpAddrCounter;
      L     #Ma.Par.ParIOByteNoCounter;
      SLD   3;
      T     #tmpAddrIO;
NETWORK
TITLE = Commands for Counter
      L     0;	// [1.8]
      L     #tmpAddrIO;	// [1.8]
      ==D;	// [1.8]
      JC    CTX0;	// [1.8]
      NOP   0;
//Clear command or counter
      A     #Ma.InPowerOk;	// [1.7]
      A     #IncCounter.OutpLOAD_VAL;	// [1.7]
      AN    #IncCounter.InpSTS_LOAD;	// [1.7]
      JC    CTJ9;	// [1.7]
      LAR1  #tmpAddrCounter;
      L     0;
      T     DID [AR1,P#4.0];
CTJ9: NOP   0;	// [1.7]
//---------------------------
      SET;
      S     #IncCounter.OutpSW_GATE;
//---------------------------
      A     #Ma.InPowerOk;
      AN    #Ma.InPowerOkDelayDone;
      O;	// [1.7]
      A     #IncCounter.OutpLOAD_VAL;	// [1.7]
      AN    #IncCounter.InpSTS_LOAD;	// [1.7]
      JCN   CTJ1;
      L     #IncCounter.VarInpHold;
      T     #IncCounter.OutpSetCount;
//    SET                               // [1.7]
      L     #IncCounter.VarInpHold;	// [1.7]
      L     #IncCounter.InpActCount;	// [1.7]
      <>D;	// [1.7]
      S     #IncCounter.OutpLOAD_VAL;
CTJ1: A     #Ma.InPowerOk;
      A     #Ma.InPowerOkDelayDone;
      AN    #IncCounter.InpSTS_LOAD;	// [1.7]
      AN    #IncCounter.OutpLOAD_VAL;	// [1.7]
      JCN   CTJ0;
      L     #IncCounter.InpActCount;
      T     #IncCounter.VarInpHold;
CTJ0: NOP   0;
      A     #IncCounter.InpSTS_LOAD;	// [1.7]
      R     #IncCounter.OutpLOAD_VAL;	// [1.7]
CTX0: NOP   0;	// [1.8]
NETWORK
TITLE = Initialisation counter module 
      L     0;	// [1.8]
      L     #tmpAddrIO;	// [1.8]
      ==D;	// [1.8]
      JC    InX0;	// [1.8]
      NOP   0;
      A     #IncCounter.InpSTS_LOAD;
      ON    #Ma.InPowerOkDelayDone;
      R     #Ma.CmdSetZeroPoint;	// [1.4]
      JC    InJ0;
//------------------------------
//When CmdSetZeroPoint then set 0
//------------------------------
      A     #Ma.CmdSetZeroPoint;
      JCN   InJ1;
      L     L#0;
      T     #IncCounter.OutpSetCount;
      T     #IncCounter.VarInpHold;	// [1.7]
      L     L#0;
      L     #Ma.OutIncrement;
      <>I;
      S     #IncCounter.OutpLOAD_VAL;	//--> Command to counter to set target value
//      SET                             // [1.4]
//      R     #Ma.CmdSetZeroPoint       // [1.4]
      L     #IncCounter.InpActCount;	// [1.4]
      L     #IncCounter.OutpSetCount;	// [1.4]
      ==D;	// [1.4]
      ON    #IncCounter.OutpLOAD_VAL;	// [1.4] //--> Command to counter to set target value
      R     #Ma.CmdSetZeroPoint;	// [1.4]
//------------------------------
//When angle >360° then set 0
//------------------------------
InJ1: L     #IncCounter.InpActCount;
      ITD;
      L     #Ma.Par.ParIncrementsPerRound;
      <=I;
      ON    #Ma.Par.ParEndless;
      JC    InJ2;
      S     #IncCounter.OutpLOAD_VAL;	//--> Command to counter to set target value
      L     L#0;
      T     #IncCounter.OutpSetCount;
      T     #IncCounter.VarInpHold;	// [1.7]
//------------------------------
//When angle < 0° then set 360°
//------------------------------
InJ2: L     #IncCounter.InpActCount;
      ITD;
      L     0;
      >=I;
      ON    #Ma.Par.ParEndless;
      JC    InJ0;
      S     #IncCounter.OutpLOAD_VAL;	//--> Command to counter to set target value
      L     #Ma.Par.ParIncrementsPerRound;
      T     #IncCounter.OutpSetCount;
      T     #IncCounter.VarInpHold;	// [1.7]
InJ0: NOP   0;
      JU    InEN;
InX0: NOP   0;	// [1.8]
//------------------------------
//When CmdSetZeroPoint then set 0
//------------------------------
      A     #Ma.CmdSetZeroPoint;	// [1.8]
      JCN   InJ7;	// [1.8]
      L     L#0;	// [1.8]
      T     #IncCounter.OutpSetCount;	// [1.8]
      T     #IncCounter.VarInpHold;	// [1.8]
      T     #Ma.OutIncrement;	// [1.8]
      T     #IncCounter.InpActCount;	// [1.8]
      L     #IncCounter.InpActCount;	// [1.8]
      L     #IncCounter.OutpSetCount;	// [1.8]
      ==D;	// [1.8]
      R     #Ma.CmdSetZeroPoint;	// [1.8]
//------------------------------
//When angle >360° then set 0
//------------------------------
InJ7: L     #IncCounter.InpActCount;	// [1.8]
      ITD;	// [1.8]
      L     #Ma.Par.ParIncrementsPerRound;	// [1.8]
      <=I;	// [1.8]
      ON    #Ma.Par.ParEndless;	// [1.8]
      JC    InJ8;	// [1.8]
      L     L#0;	// [1.8]
      T     #IncCounter.OutpSetCount;	// [1.8]
      T     #IncCounter.VarInpHold;	// [1.8]
      T     #IncCounter.InpActCount;	// [1.8]
//------------------------------
//When angle < 0° then set 360°
//------------------------------
InJ8: L     #IncCounter.InpActCount;	// [1.8]
      ITD;	// [1.8]
      L     0;	// [1.8]
      >=I;	// [1.8]
      ON    #Ma.Par.ParEndless;	// [1.8]
      JC    InJ9;	// [1.8]
      L     #Ma.Par.ParIncrementsPerRound;	// [1.8]
      T     #IncCounter.OutpSetCount;	// [1.8]
      T     #IncCounter.VarInpHold;	// [1.8]
      T     #IncCounter.InpActCount;	// [1.8]
InJ9: NOP   0;	// [1.8]
InEN: NOP   0;	// [1.8]
NETWORK
TITLE = Read Global Command
      A     "GCS7_Gr_OutFaultReset";	// OutFaultReset
      S     #Ma.CmdFaultReset;
NETWORK
TITLE = Write Outputs of counter
      L     0;
//    L     #tmpAddrCounter             // [1.8]
      L     #tmpAddrIO;	// [1.11]
      ==D;
      JC    WCJ0;
///Write Outputs  Counter left
      LAR1  #tmpAddrCounter;
      L     DID [AR1,P#0.0];
      LAR1  #tmpAddrIO;
      T     PQD [AR1,P#0.0];
      LAR1  #tmpAddrCounter;
      L     DID [AR1,P#4.0];
      LAR1  #tmpAddrIO;
      T     PQD [AR1,P#4.0];
WCJ0: NOP   0;
NETWORK
TITLE = Read Counter
      L     0;
//      L     #tmpAddrCounter   // JV [1.3]
      L     #tmpAddrIO;	// JV [1.3]
      ==D;
      JC    RCJ0;
//Read IO Counter left
      LAR1  #tmpAddrIO;
      L     PID [AR1,P#0.0];
      LAR1  #tmpAddrCounter;
      T     DID [AR1,P#8.0];
      LAR1  #tmpAddrIO;
      L     PID [AR1,P#4.0];
      LAR1  #tmpAddrCounter;
      T     DID [AR1,P#12.0];
RCJ0: NOP   0;
NETWORK
TITLE = Speed monitoring
      NOP   0;
//==========================================================
//Speed Monitoring Left
//==========================================================
//- Check if increment is changing
      A(;
      L     #IncCounter.InpActCount;
      ITD;
      L     #Ma.OutIncrement;
      ==D;
      );
      A(;
      O     #Motor.OutpRunFwd;
      O     #Motor.OutpRunRev;
      );
      AN    #Ma.CmdFaultReset;
      JC    M1J1;
      L     #Ma.Par.ParMonTime;	//5s
      T     #Ma.Par.OutMonTime;
      S     #SM.InpTrue;
//---Run monitoring time
M1J1: AN    "GCS7_Gr_OutTick200ms";
      JC    M1J2;
      L     #Ma.Par.OutMonTime;
      +     -2;
      T     #Ma.Par.OutMonTime;
      L     0;
      >=I;
      JC    M1J2;
      T     #Ma.Par.OutMonTime;
      R     #SM.InpTrue;
//---Store old counter value
M1J2: L     #IncCounter.InpActCount;
      ITD;
      T     #Ma.OutIncrement;
NETWORK
TITLE = Calculation position
      NOP   0;
//-----
      L     3.600000e+03;
      L     #Ma.Par.ParIncrementsPerRound;
      DTR;
      /R;
      L     #Ma.OutIncrement;
      DTR;
      TAK;
      *R;
      RND;
      T     #Ma.OutPositionAngle;	//Position [0.1°]
//--------
      L     1.000000e+03;
      L     #Ma.Par.ParIncrementsPerRound;
      DTR;
      /R;
      L     #Ma.OutIncrement;
      DTR;
      TAK;
      *R;
//      TRUNC 
      RND;
      T     #Ma.OutPositionRel;	//Position [0.1%]
NETWORK
TITLE = Check Adjusted
//Test is actual prosition is in range:
//    InPositionTarget+Ma.Par.ParTolPosition  OutPositionLeft
      NOP   0;
//------------------
      L     #Ma.OutPositionAngle;
      L     #Ma.InPositionTarget;
      -I;
      JP    A1J1;
      NEGI;
A1J1: T     #tmpAngle1;
      L     1800;
      <=I;
      ON    #Ma.Par.ParEndless;
      TAK;
      JC    A1J2;
      L     3600;
      L     #tmpAngle1;
      -I;
A1J2: L     #Ma.Par.ParTolPosition;
      <=I;
      =     #Ma.OutAdjusted;
      A     #Ma.OutAdjusted;
      A     #Ma.InAdjusting;
      =     #tmpAdjusted;
NETWORK
TITLE = Round counter
      L     0;	//[1.9]
      L     #tmpAddrIO;	//[1.9]
      ==D;	//[1.9]
      JCN   rcj0;	//[1.9]
      AN    #Ma.Par.ParEndless;	//[1.9]
      JC    rcj9;	//[1.9]
      AN    #Ma.CmdNewJob;
      JC    rcj1;	//[1.9]
      S     #Ma.OutEdgeCntRoundFwd;
      S     #Ma.OutEdgeCntRoundRev;
      R     #Ma.CmdNewJob;
      L     0;
      T     #Ma.OutCntRound;
      T     #Ma.OutPositionStart;
rcj1: NOP   0;
//------------------
//Calculate Delta angel between OutStartPosition and OutPositionAngle 
//------------------
      L     #Ma.OutPositionAngle;
      L     #Ma.OutPositionStart;
      -I;
      JP    rcj2;	//[1.9]
      NEGI;
rcj2: T     #tmpAngle1;
      L     1800;
      <=I;
      TAK;
      JC    rcj3;	//[1.9]
      L     3600;
      L     #tmpAngle1;
      -I;
rcj3: T     #tmpAngleDelta;
      L     1700;	//Delta angle 170°
      >I;
      R     #Ma.OutEdgeCntRoundFwd;
      R     #Ma.OutEdgeCntRoundRev;
//----------------------                
//Round Counter                         
//---------------------                 
      A(;
      L     #tmpAngleDelta;
      L     #Ma.Par.ParTolPosition;	//[1.1]Delta angle 1°
      <=I;
      );
      JCN   rcj9;	//[1.9]
      AN    #Ma.StStartedFwd;
      AN    #Motor.InEnableFwd;
      JC    rcj4;	//[1.9]
      A     #Ma.OutEdgeCntRoundFwd;
      JC    rcj9;	//[1.9]
      S     #Ma.OutEdgeCntRoundFwd;
      R     #Ma.OutEdgeCntRoundRev;
      L     #Ma.OutCntRound;
      L     L#1;
      +D;
      T     #Ma.OutCntRound;
      JU    rcj9;	//[1.9]
rcj4: AN    #Ma.StStartedRev;	//[1.9]
      AN    #Motor.InEnableRev;	//[1.9]
      JC    rcj9;	//[1.9]
      A     #Ma.OutEdgeCntRoundRev;
      JC    rcj9;	//[1.9]
      S     #Ma.OutEdgeCntRoundRev;
      R     #Ma.OutEdgeCntRoundFwd;
      L     #Ma.OutCntRound;
      L     L#1;
      -D;
      T     #Ma.OutCntRound;
      L     0;
      >=D;
      JC    rcj9;	//[1.9]
      L     0;
      T     #Ma.OutCntRound;
rcj9: NOP   0;	//[1.9]
      JU    RCJ9;	//[1.9]
rcj0: NOP   0;	//[1.9]
      AN    #Ma.Par.ParEndless;	//[1.2]
      JC    RCJ9;	//[1.2]
      AN    #Ma.CmdNewJob;
      JC    RCJ1;
      S     #Ma.OutEdgeCntRoundFwd;	//[1.1]
      S     #Ma.OutEdgeCntRoundRev;	//[1.1]
      R     #Ma.CmdNewJob;
      L     0;
      T     #Ma.OutCntRound;
//      L     #Ma.OutPositionAngle    //[1.5]  // UK 9.11.2006 geändert
      T     #Ma.OutPositionStart;
RCJ1: NOP   0;
//------------------
//Calculate Delta angel between OutStartPosition and OutPositionAngle 
//------------------
      L     #Ma.OutPositionAngle;
      L     #Ma.OutPositionStart;
      -I;
      JP    RCJ2;
      NEGI;
RCJ2: T     #tmpAngle1;
      L     1800;
      <=I;
      TAK;
      JC    RCJ3;
      L     3600;
      L     #tmpAngle1;
      -I;
RCJ3: T     #tmpAngleDelta;
      L     1700;	//Delta angle 170°
      >I;
      R     #Ma.OutEdgeCntRoundFwd;	//[1.1]
      R     #Ma.OutEdgeCntRoundRev;	//[1.1]
//----------------------                //[1.1]
//Round Counter                         //[1.1]
//---------------------                 //[1.1]
      A(;	//[1.1]
      L     #tmpAngleDelta;	//[1.1]
      L     #Ma.Par.ParTolPosition;	//[1.1]Delta angle 1°
      <=I;	//[1.1]
      );	//[1.1]
      JCN   RCJ9;	//[1.1]
//      UN    #Ma.StStartedFwd            //[1.2]
//      UN    #Motor.InEnableFwd          //[1.1]
      AN    #IncCounter.InpSTS_C_UP;	//[1.6]       UK 23.11.2006 geändert
      JC    RCJ4;	//[1.1]
      A     #Ma.OutEdgeCntRoundFwd;	//[1.1]
      JC    RCJ9;	//[1.1]
      S     #Ma.OutEdgeCntRoundFwd;	//[1.1]
      R     #Ma.OutEdgeCntRoundRev;	//[1.1]
      L     #Ma.OutCntRound;	//[1.1]
//      +     L#1                         //[1.1]  // UK 14.11.2006 geändert
      L     L#1;	//[1.5]       UK 14.11.2006 geändert
      +D;	//[1.5]       UK 14.11.2006 geändert
      T     #Ma.OutCntRound;	//[1.1]
      JU    RCJ9;	//[1.1]
// RCJ4: UN    #Ma.StStartedRev            //[1.2]
// RCJ4: UN    #Motor.InEnableRev          //[1.1]
RCJ4: AN    #IncCounter.InpSTS_C_DN;	//[1.6]       UK 23.11.2006 geändert
      JC    RCJ9;	//[1.1]
      A     #Ma.OutEdgeCntRoundRev;	//[1.1]
      JC    RCJ9;	//[1.1]
      S     #Ma.OutEdgeCntRoundRev;	//[1.1]
      R     #Ma.OutEdgeCntRoundFwd;	//[1.1]
      L     #Ma.OutCntRound;	//[1.1]
      L     L#1;	//[1.1]
      -D;	//[1.1]
      T     #Ma.OutCntRound;	//[1.1]
      L     0;	//[1.1]
      >=D;	//[1.1]
      JC    RCJ9;	//[1.1]
      L     0;	//[1.1]
      T     #Ma.OutCntRound;	//[1.1]
RCJ9: NOP   0;
NETWORK
TITLE = Interlocking
//===Global Group Orders===
      A     "GCS7_Gr_OutManualOff";	//Gr.OutManualOff
      R     #Ma.InManual;
      A     #Ma.InManual;
      S     "GCS7_Gr_InManual";	//Gr.InManual
//--------------
      A     #Ma.CmdOnFwd;
      S     #Ma.OutManStartReqFwd;
      R     #Ma.OutManStartReqRev;
      A     #Ma.CmdOnRev;
      R     #Ma.OutManStartReqFwd;
      S     #Ma.OutManStartReqRev;
      A     #Ma.CmdOff;
      ON    #Ma.InManual;
      R     #Ma.OutManStartReqFwd;
      R     #Ma.OutManStartReqRev;
//--- Fault----
      A     #Motor.StFault;
      O     #Speed.StFault;
      O     #LSZeroPoint.StFault;
      O     #Product.StFault;
      O     #SM.StFault;
      =     #tmpFaultSum;
//--- InLocal----
      A     #Ma.InLocal;
      AN    #Ma.InManual;
      =     #tmpLocal;
      =     #Motor.InLocal;
      =     #Speed.InLocal;
      =     #LSZeroPoint.InLocal;
      =     #Product.InLocal;
      =     #SM.InLocal;
//--- Fault Reset -------------
      A     #Ma.CmdFaultReset;
      S     #Motor.CmdFaultReset;
      S     #Speed.CmdFaultReset;
      S     #LSZeroPoint.CmdFaultReset;
      S     #Product.CmdFaultReset;
      S     #SM.CmdFaultReset;
NETWORK
TITLE = Interlocking Motor
      AN    #tmpFaultSum;
      ON    #Ma.InInterlocked;
      A(;
      AN    #tmpAdjusted;
      ON    #Ma.InAdjusting;
      AN    #Ma.InManual;
      O     #Ma.OutManStartReqRev;
      );
      A     #Ma.InEnableRev;
      A     #Ma.InPowerOkDelayDone;
      =     #Motor.InEnableRev;
      AN    #tmpFaultSum;
      ON    #Ma.InInterlocked;
      A(;
      AN    #tmpAdjusted;
      ON    #Ma.InAdjusting;
      AN    #Ma.InManual;
      O     #Ma.OutManStartReqFwd;
      );
//      U(                                //[1.2]
//      U     #Ma.InLoading               //[1.2]
//      U     #Product.InpTrue            //[1.2]
//      ON    #Ma.InLoading               //[1.2]
//      )                                 //[1.2]
      A(;	//[1.10]
      A     #Product.StCtoTrue;	//[1.10]
      O     #Product.StTrue;	//[1.10]
      A     #Ma.InLoading;	//[1.10]
      O;	//[1.10]
      AN    #Ma.InLoading;	//[1.10]
      );	//[1.10]
      A     #Ma.InEnableFwd;
      A     #Ma.InPowerOkDelayDone;
      =     #Motor.InEnableFwd;
      A     #Ma.CmdNext;
      O     #Ma.InManual;
      S     #Motor.CmdNext;
NETWORK
TITLE = Interlocking Speed
      AN    #Motor.InEnableRev;
      AN    #Motor.InEnableFwd;
      AN    #Ma.InManual;
      AN    #Motor.InManual;
      A     "SYS_infLog0";	// never disable JV [1.3]
      =     #Speed.InDisable;
      L     0;
      JC    SpJ1;
      L     #Ma.InSpeed;
SpJ1: T     #Speed.InOutValuePc;
      SET;
      =     #Speed.Par.ParValuePc;
NETWORK
TITLE = Interlocking Flow control
//At start of loading:
//   If the flow detector is covered then generate alarm
//
//During loading:
//   If the flowdectecor is to long covered then generate alarm
      CLR;
      =     #Product.InMonTrue;
      =     #Product.Par.Par2WorkingCond;
      A     #Ma.InLoading;
      =     #Product.InMonFalse;
      A     #Product.InpTrue;
      FP    #Ma.OutEdgeLoading;
      S     #Product.CmdRunTimeoutTime;
NETWORK
TITLE = Control Element SM
      A     #Motor.StStartedRev;
      O     #Motor.StStartedFwd;
      =     #SM.InMonTrue;
NETWORK
TITLE = Control Element LSZeroPoint
//      CLR   
//      =     #LSZeroPoint.InpTrue
//      =     #LSZeroPoint.InMonTrue
      A     #Ma.InManual;
      O     #Motor.InManual;
      A     #LSZeroPoint.OutFlagPos;
      S     #Motor.CmdOff;
NETWORK
TITLE = Call Motor
      CALL  #Motor;
NETWORK
TITLE = Call Analog Output: Speed
      CALL  #Speed;
NETWORK
TITLE = Call Digital Input: LSZeroPoint
      CALL  #LSZeroPoint;
NETWORK
TITLE = Call Digital Input: Product
      CALL  #Product;
NETWORK
TITLE = Call Digital Input: SM
      CALL  #SM;
NETWORK
TITLE = States
      A     #Ma.StStopped;
      JC    S0;
      A     #Ma.StAdjusted;
      JC    S6;
      A     #Ma.StStartedFwd;
      JC    S2;
      A     #Ma.StStartedRev;
      JC    S5;
      A     #Ma.StStopping;
      JC    S3;
      A     #Ma.StStarting;
      JC    S1;
      A     #Ma.StFault;
      JC    S4;
      JU    xxS0;	//Initialise: goto StStopped
NETWORK
TITLE = StStopped
xxS0: S     #Ma.StStopped;
      JU    SAVE;
//---Transition -> StFault
S0:   A     #tmpFaultSum;
      R     #Ma.StStopped;
      JC    xxS4;
//---Transition -> StStarting
      A     #Ma.OutManStartReqFwd;
      O     #Ma.OutManStartReqRev;
      A     #Ma.InManual;
      ON    #Motor.StStopped;
      R     #Ma.StStopped;
      JC    xxS1;
//---Transition for StAdjusted
      A     #tmpAdjusted;
      AN    #tmpLocal;
      R     #Ma.StStopped;
      JC    xxS6;
      JU    SAVE;
NETWORK
TITLE = StStarting
//== Any transition to StStarting
xxS1: SET;
      S     #Ma.StStarting;
      JU    SAVE;
//== Logic ====
//---Transition -> StFault
S1:   A     #tmpFaultSum;
      R     #Ma.StStarting;
      JC    xxS4;
//---Transition -> StStartedUn
      A     #Motor.StStartedFwd;
      R     #Ma.StStarting;
      JC    xxS2;
//---Transition -> StStartingRev
      A     #Motor.StStartedRev;
      R     #Ma.StStarting;
      JC    xxS5;
//---Transition for StStopping
      A     #Motor.StStopped;
      AN    #Ma.OutManStartReqFwd;
      AN    #Ma.OutManStartReqRev;
      O     #tmpLocal;
      R     #Ma.StStarting;
      JC    xxS3;
//---Transition for StAdjusted
      A     #tmpAdjusted;
      AN    #tmpLocal;
      R     #Ma.StStarting;
      JC    xxS6;
      JU    SAVE;
NETWORK
TITLE = StStartedFwd
xxS2: SET;
      S     #Ma.StStartedFwd;
      JU    SAVE;
//---Transition -> StFault
S2:   A     #tmpFaultSum;	//---Condition for StFault
      R     #Ma.StStartedFwd;
      JC    xxS4;
//---Transition -> StStoppting
      AN    #Motor.StStartedFwd;
      R     #Ma.StStartedFwd;
      JC    xxS3;
      JU    SAVE;
NETWORK
TITLE = StStartedRev
xxS5: SET;
      S     #Ma.StStartedRev;
      JU    SAVE;
//---Transition -> StFault
S5:   A     #tmpFaultSum;	//---Condition for StFault
      R     #Ma.StStartedRev;
      JC    xxS4;
//---Transition -> StStoppting
      AN    #Motor.StStartedRev;
      R     #Ma.StStartedRev;
      JC    xxS3;
      JU    SAVE;
NETWORK
TITLE = StAdjusted
xxS6: SET;
      S     #Ma.StAdjusted;
//---Transition -> StFault
S6:   A     #tmpFaultSum;
      R     #Ma.StAdjusted;
      JC    xxS4;
//---Transition for StStarting
      AN    #Motor.StStopped;
      R     #Ma.StAdjusted;
      JC    xxS1;
//---Transition -> StStopping
      AN    #tmpAdjusted;
      O     #tmpLocal;
      R     #Ma.StAdjusted;
      JC    xxS3;
      JU    SAVE;
NETWORK
TITLE = StStopping
//===Any transition to StStopping
xxS3: SET;
      S     #Ma.StStopping;
      JU    SAVE;
//===Logic =======================
//---Transtition -> StFault
S3:   A     #tmpFaultSum;
      R     #Ma.StStopping;
      JC    xxS4;
//---Transition for StAdjusted
      A     #tmpAdjusted;
      A     #Motor.StStopped;
      AN    #tmpLocal;	// [1.2]
      R     #Ma.StStopping;
      JC    xxS6;
//---Transition -> StStopped
      A     #Motor.StStopped;
      R     #Ma.StStopping;
      JC    xxS0;
//---Transition -> StStarting
      AN    #Motor.StStopping;
      R     #Ma.StStopping;
      JC    xxS1;
      JU    SAVE;
NETWORK
TITLE =  StFault
// Any transiton to Fault  
xxS4: SET;
      S     #Ma.StFault;
//===logic
//---Transition -> StStopping
S4:   AN    #tmpFaultSum;
      R     #Ma.StFault;
      JC    xxS3;
      JU    SAVE;
NETWORK
TITLE = Global End
SAVE: SET;	//---Clear all commands
      R     #Ma.CmdOnFwd;
      R     #Ma.CmdOnRev;
      R     #Ma.CmdOff;
      R     #Ma.CmdNext;
      R     #Ma.CmdFaultReset;
//---------------------------------
      AN    #Motor.StStarting;
      AN    #Motor.StStartedFwd;
      AN    #Motor.StStartedRev;
      ON    #Ma.InManual;
      R     #Ma.OutManStartReqRev;
      R     #Ma.OutManStartReqFwd;
NETWORK
TITLE = State Code
//--Stopped, Substate ---
      A     #Ma.StStopped;
      L     1;
      JC    STC9;
      A     #Ma.StStarting;
      L     2;
      JC    STC9;
      A     #Ma.StStartedFwd;
      L     3;
      JC    STC9;
      A     #Ma.StStartedRev;
      L     5;
      JC    STC9;
      A     #Ma.StAdjusted;
      L     6;
      JC    STC9;
      A     #Ma.StStopping;
      L     7;
      JC    STC9;
      L     32;	// Code: fault
STC9: L     #Ma.StCode;	// Old state code
      TAK;
      T     #Ma.StCode;	// Save state code
      <>I;
      L     3;	// Load code for CBit methode
      CC    "SYS_CBitCtrl";
END_FUNCTION_BLOCK

FUNCTION_BLOCK "GCS7_M_Roll8Stand_DP"	// FB 87
TITLE = Roll stand with 8
//  
//COPYRIGHT:    (C) 1997  BUHLER AG, CH-9240 UZWIL,  SWITZERLAND
//
//PRODUCT:      GCS7
//
//TITLE:        FB 87 Machine roll stand with 8 rolls with MDDR/T
//
//REVISION:     11
//
//-------------------------------------------------------------------------
//
//IDENT:        AUTHOR:             DEPT:                       DATE:
//
//FB87.6.1      A. Egli             CT3                         03-Mar-2008
//              - Condition OutStartupDone 
//              - No stop motors if HLOutlet is covered
//FB87.6.0      A. Egli             CT3                         22-Feb-2008
//              HLOutlet3SideX instead of SM2SideX
//FB87.5.2      A. Egli             CT3                         14-Feb-2008
//              MDDR/T: Manual Motor interlocke with Status.SxEnableMotors
//FB46.5.1      A. Egli             CT3                         10-Oct-2007
//              Condition Stopped if only one motor
//FB46.5.0      A. Egli             CT3                         06-Apr-2007
//              New Release R2 
//FB46.4.2      A. Egli             CT3                         05-Mai-2004
//              CmdOff in manual mode
//FB46.4.1      A. Egli             CT3                         23-Sep-2003
//              InEnable=0 must stop motor when ParManual=1 and InManual=0
//FB46.4.0      A. Egli             CT3                         18-Oct-2002
//              New Release with one block 
//FB46.3.2      A. Egli             CT3                         18-Okt-2002
//              Condition tmpStarted with ParMa.Par4Rolls=0 
//FB46.3.1      A. Egli             CT3                         08-Feb-2000
//              Condition Monitoring HL 
//FB46.3.0      A. Egli             CT3                         11-Oct-1999
//              Local data reduced 
//FB46.2B       K. Tischer          MU664                       06-Mrz-1999
//              CC FC2 not UC FC2
//FB46.2A       A. Egli             CT3                         04-Mai-1998
//              StFault = StCode 32
//FB46.1A       A.Egli              AEE61                       12-Nov-1997
//              1st Release in S7
//
//-------------------------------------------------------------------------
//
//PURPOSE:      MANUAL : see [SSW-MA-Roll8Stand_MAN_en]
//
//RESTRICTIONS: S7
//
//-------------------------------------------------------------------------
//
//
AUTHOR : EA
FAMILY : GCS7LL
NAME : Rolls8
VERSION : 6.1
VAR
  Ma : UDT 20870;
  MotorLowSide1 : FB 12;	//Element
  MotorLowSide2 : FB 12;	//Element
  SM1Side1 : FB 14;	//Element
  SM1Side2 : FB 14;	//Element
  HLInletSide1 : FB 14;	//Element
  HLInletSide2 : FB 14;	//Element
  HLBackupLeftSide1 : FB 14;	//Element Only 8 with 8 rolls
  HLBackupLeftSide2 : FB 14;	//Element Only 8 with 8 rolls
  MotorUpSide1 : FB 12;	//Element
  MotorUpSide2 : FB 12;	//Element
  HLOutlet3Side1 : FB 14;	//Element
  HLOutlet3Side2 : FB 14;	//Element
  HLBackupRightSide1 : FB 14;	//Element Only 8 with 8 rolls
  HLBackupRightSide2 : FB 14;	//Element Only 8 with 8 rolls
  HLInletSide1Div : FB 14;	//Element Only if side 1 is divided (Side 1 left)
  HLInletSide2Div : FB 14;	//Element Only if side 2 is divided (Side 2 left)
  MDDx : FB 37;
  FeedrollSide1 : FB 17;
  FeedrollSide2 : FB 17;
  FeedrollSide1Div : FB 17;
  FeedrollSide2Div : FB 17;
  HLOutlet1Side1 : FB 14;	//Element
  HLOutlet2Side1 : FB 14;	//Element
  HLOutlet1Side2 : FB 14;	//Element
  HLOutlet2Side2 : FB 14;	//Element
END_VAR
VAR_TEMP
  tmpFaultSum : BOOL ;
  tmpWarning : BOOL ;
  tmpStarted : BOOL ;
  tmpNext : BOOL ;
  tmpLocal : BOOL ;
  tmpEnable : BOOL ;
  tmpSeqStop : BOOL ;
END_VAR
BEGIN
NETWORK
TITLE = PC Control
//=== Test Object number =====================
      L     "SYS_DirectCtrlDB".PC.ObjectNo;	//PCControl.ObjectNo
      L     #Ma.Par.ParObjectNo;	//Input ObjectNo    
      <>I;
      JC    aEnd;
//=== Test OType      ========================
      L     2087;	//Input object type
      L     "SYS_DirectCtrlDB".PC.ObjectType;	//PCControl.ObjectType
      <>I;
      JC    aEnd;
//=== Test Handshake =========================
      A     "SYS_DirectCtrlDB".PC.Hsk.FExamine;	// Handshake.FExamine
      JC    aExa;
      A     "SYS_DirectCtrlDB".PC.Hsk.FDefineCmd;	// Handshake.FDefineCmd
      O     "SYS_DirectCtrlDB".PC.Hsk.FDefinePara;	// Handshake.FDefinePara
      JC    aCmd;
      JU    aIni;
aIni: L     2;	// FcInit
      UC    "SYS_DirectCtrl";
      JU    aEnd;
// Write new commands from PC to Interface of group 
aCmd: A     "SYS_DirectCtrlDB".PC.Cmd1[0];	//InEnableDosingOn
      S     #Ma.InEnableDosing;
      A     "SYS_DirectCtrlDB".PC.Cmd2[10];	//InEnableDosingOff
      R     #Ma.InEnableDosing;
      A     "SYS_DirectCtrlDB".PC.Cmd1[1];	//CmdEnableSide1
      R     #Ma.InDisableSide1;
      A     "SYS_DirectCtrlDB".PC.Cmd2[1];	//CmdDisableSide1
      S     #Ma.InDisableSide1;
      A     "SYS_DirectCtrlDB".PC.Cmd1[2];	//CmdEnableSide2
      R     #Ma.InDisableSide2;
      A     "SYS_DirectCtrlDB".PC.Cmd2[2];	//CmdDisableSide2
      S     #Ma.InDisableSide2;
      A     "SYS_DirectCtrlDB".PC.Cmd1[3];	//CmdOverwriteHLOn
      S     #Ma.InOverrideHL;
      A     "SYS_DirectCtrlDB".PC.Cmd2[3];	//CmdOverwriteHLOff
      R     #Ma.InOverrideHL;
      A     "SYS_DirectCtrlDB".PC.Cmd1[4];	//CmdRestDischargeOn
      S     #Ma.InRestDischarge;
      A     "SYS_DirectCtrlDB".PC.Cmd2[4];	//CmdRestDischargeOff
      R     #Ma.InRestDischarge;
      A     "SYS_DirectCtrlDB".PC.Cmd1[8];	//Cmd1[8]=CmdOff
      S     #Ma.CmdOff;
      A     "SYS_DirectCtrlDB".PC.Cmd1[9];	//Cmd1[9]=CmdOn
      S     #Ma.CmdOn;
      A     "SYS_DirectCtrlDB".PC.Cmd1[10];	//Cmd1[10]=CmdNext
      S     #Ma.CmdNext;
      A     "SYS_DirectCtrlDB".PC.Cmd1[11];	//Cmd1[11]=CmdFaultReset
      S     #Ma.CmdFaultReset;
      A     "SYS_DirectCtrlDB".PC.Cmd1[13];	//Cmd1[13]=CmdManualOn
      S     #Ma.InManual;
      A     "SYS_DirectCtrlDB".PC.Cmd2[13];	//Cmd1[13]=CmdManualOff
      R     #Ma.InManual;
//-----------------------------------------------------------
//Audit Log
aExa: NOP   0;
      TAR2;	// Address Dynamic datas
      T     "SYS_DirectCtrlDB".GC.InDynAddr;	// -->PCControl.GC.InDynAddr
      L     14;	// Length Dynamic data
      T     "SYS_DirectCtrlDB".GC.InDynLen;	// -->PCControl.GC.InDynLen
      L     0;
      T     "SYS_DirectCtrlDB".GC.InParaAddr;	// -->PCControl.GC.InParaAddr
      T     "SYS_DirectCtrlDB".GC.InParaLen;	// -->PCControl.GC.InParaLen
      L     1;	// Code FcExamine
      UC    "SYS_DirectCtrl";
      L     11;	//Revision
      T     "SYS_DirectCtrlDB".GC.Revision;
//------------------------------------------
aEnd: NOP   0;
NETWORK
TITLE = Interlocking
//===Global Group Orders===
      A     "GCS7_Gr_OutManualOff";	//Gr.OutManualOff
      R     #Ma.InManual;
      A     #Ma.InManual;
      S     "GCS7_Gr_InManual";	//Gr.InManual
// temporare
      AN    #Ma.StStarting;
      ON    #Ma.InManual;
      O     #Ma.CmdOff;	//[4.2]
      R     #Ma.OutStartMan;
      O     #Ma.CmdOn;
      S     #Ma.OutStartMan;
      A     #Ma.CmdNext;
      AN    #Ma.InManual;
      O     #Ma.OutStartMan;
      =     #tmpNext;
      A     #Ma.InManual;
      ON    #Ma.InLocal;
      A(;
      A     #Ma.Par.ParManual;	//[4.1]
      A     #Ma.InManual;
      O     #Ma.InEnable;
      );
      A(;
      AN    #MDDx.StFault;
      ON    #Ma.Par.ParWithMDDx;
      );
      AN    #Ma.CmdOff;
      =     #tmpEnable;
      A     #Ma.InSeqStop;
      AN    #Ma.InManual;
      =     #tmpSeqStop;
//Warning
      A     #HLInletSide1.StTrue;
      O     #HLInletSide2.StTrue;
      O     #HLInletSide1Div.StTrue;
      O     #HLInletSide2Div.StTrue;
      A     #Ma.InOverrideHL;
      O     #MDDx.OutWarning;
      =     #tmpWarning;
      =     #Ma.OutWarning;
//--- Fault----
      A     #MotorLowSide1.StFault;
      O     #MotorUpSide1.StFault;
      O     #MotorLowSide2.StFault;
      O     #MotorUpSide2.StFault;
      O     #HLBackupLeftSide1.StFault;
      O     #HLBackupLeftSide2.StFault;
      O     #HLBackupRightSide1.StFault;
      O     #HLBackupRightSide2.StFault;
      O     #HLInletSide1.StFault;
      O     #HLInletSide2.StFault;
      O     #HLInletSide1Div.StFault;
      O     #HLInletSide2Div.StFault;
      O     #SM1Side1.StFault;
      O     #SM1Side2.StFault;
      O     #HLOutlet3Side1.StFault;
      O     #HLOutlet3Side2.StFault;
      O     #MDDx.StFault;
      O     #MDDx.OutFaultRelevant;
      O     #FeedrollSide1.StFault;
      O     #FeedrollSide2.StFault;
      O     #FeedrollSide1Div.StFault;
      O     #FeedrollSide2Div.StFault;
      O     #HLOutlet1Side1.StFault;
      O     #HLOutlet2Side1.StFault;
      O     #HLOutlet1Side2.StFault;
      O     #HLOutlet2Side2.StFault;
      =     #tmpFaultSum;
//--- Local mode --
      A     #Ma.InLocal;
      AN    #Ma.InManual;
      =     #tmpLocal;
      =     #MotorLowSide1.InLocal;
      =     #MotorLowSide2.InLocal;
      =     #SM1Side1.InLocal;
      =     #SM1Side2.InLocal;
      =     #MotorUpSide1.InLocal;
      =     #MotorUpSide2.InLocal;
      =     #MDDx.InLocal;
      =     #FeedrollSide1.InLocal;
      =     #FeedrollSide2.InLocal;
      =     #FeedrollSide1Div.InLocal;
      =     #FeedrollSide2Div.InLocal;
      A     #Ma.InDisableSide1;
      A     #MotorLowSide1.StStopped;
      O     #tmpLocal;
      =     #HLInletSide1.InLocal;
      =     #HLOutlet1Side1.InLocal;
      =     #HLOutlet2Side1.InLocal;
      =     #HLOutlet3Side1.InLocal;	//[6.0]
      =     #HLBackupLeftSide1.InLocal;
      =     #HLBackupRightSide1.InLocal;
      =     #HLInletSide1Div.InLocal;
      A     #Ma.InDisableSide2;
      A     #MotorLowSide2.StStopped;
      O     #tmpLocal;
      =     #HLInletSide2.InLocal;
      =     #HLBackupLeftSide2.InLocal;
      =     #HLBackupRightSide2.InLocal;
      =     #HLOutlet1Side2.InLocal;
      =     #HLOutlet2Side2.InLocal;
      =     #HLOutlet3Side2.InLocal;	//[6.0]
      =     #HLInletSide2Div.InLocal;
//--- Fault Reset -------------
      A     #Ma.CmdFaultReset;
      S     #MotorLowSide1.CmdFaultReset;
      S     #MotorLowSide2.CmdFaultReset;
      S     #SM1Side1.CmdFaultReset;
      S     #SM1Side2.CmdFaultReset;
      S     #HLInletSide1.CmdFaultReset;
      S     #HLInletSide2.CmdFaultReset;
      S     #HLBackupLeftSide1.CmdFaultReset;
      S     #HLBackupLeftSide2.CmdFaultReset;
      S     #MotorUpSide1.CmdFaultReset;
      S     #MotorUpSide2.CmdFaultReset;
      S     #HLOutlet3Side1.CmdFaultReset;
      S     #HLOutlet3Side2.CmdFaultReset;
      S     #HLBackupRightSide1.CmdFaultReset;
      S     #HLBackupRightSide2.CmdFaultReset;
      S     #HLInletSide1Div.CmdFaultReset;
      S     #HLInletSide2Div.CmdFaultReset;
      S     #MDDx.CmdFaultReset;
      S     #FeedrollSide1.CmdFaultReset;
      S     #FeedrollSide2.CmdFaultReset;
      S     #FeedrollSide1Div.CmdFaultReset;
      S     #FeedrollSide2Div.CmdFaultReset;
      S     #HLOutlet1Side1.CmdFaultReset;
      S     #HLOutlet2Side1.CmdFaultReset;
      S     #HLOutlet1Side2.CmdFaultReset;
      S     #HLOutlet2Side2.CmdFaultReset;
//==== Monitoring ================
//  --HL Backup
      A     #MDDx.Side1.Out.OutLCAlarm.A064HLBackupLeft;
      ON    #Ma.Par.ParWithMDDx;
      AN    #Ma.Par.Par4Rolls;
      =     #HLBackupLeftSide1.InMonFalse;
      A     #MDDx.Side2.Out.OutLCAlarm.A064HLBackupLeft;
      ON    #Ma.Par.ParWithMDDx;
      AN    #Ma.Par.Par4Rolls;
      =     #HLBackupLeftSide2.InMonFalse;
      A     #MDDx.Side1.Out.OutLCAlarm.A066HLBackupRight;
      ON    #Ma.Par.ParWithMDDx;
      AN    #Ma.Par.Par4Rolls;
      =     #HLBackupRightSide1.InMonFalse;
      A     #MDDx.Side2.Out.OutLCAlarm.A066HLBackupRight;
      ON    #Ma.Par.ParWithMDDx;
      AN    #Ma.Par.Par4Rolls;
      =     #HLBackupRightSide2.InMonFalse;
//  --HL Inlet
      AN    #Ma.InOverrideHL;
      =     #HLInletSide1.InMonFalse;
      =     #HLInletSide2.InMonFalse;
      =     #HLInletSide1Div.InMonFalse;
      =     #HLInletSide2Div.InMonFalse;
//  --HLOutlet
      SET;
      =     #HLOutlet1Side1.InMonFalse;
      =     #HLOutlet2Side1.InMonFalse;
      =     #HLOutlet3Side1.InMonFalse;	//[6.0]
      =     #HLOutlet1Side2.InMonFalse;
      =     #HLOutlet2Side2.InMonFalse;
      =     #HLOutlet3Side2.InMonFalse;	//[6.0]
//  --SM Side 1
      AN    #Ma.Par.ParWithMDDx;
      A     #Ma.InpPressureSide1;
      =     #SM1Side1.InMonTrue;
//  --SM Side 2
      AN    #Ma.Par.ParWithMDDx;
      A     #Ma.InpPressureSide2;
      =     #SM1Side2.InMonTrue;
NETWORK
TITLE = Interlocking Motors Rolls
      A     #MDDx.Status.S1EnableMotors;
      ON    #Ma.Par.ParWithMDDx;
      A     #tmpNext;
      S     #MotorLowSide1.CmdNext;
      S     #MotorUpSide1.CmdNext;
      A     #Ma.Par.Par4Rolls;
      ON    #Ma.Par.ParWithMotorUpSide1;	//[5.1]
      A     #MotorLowSide1.StStartedFwd;
      O     #MotorUpSide1.StStartedFwd;
      O     #Ma.InDisableSide1;
      A(;
      A     #MDDx.Status.S2EnableMotors;
      ON    #Ma.Par.ParWithMDDx;
      );
      A     #tmpNext;
      S     #MotorLowSide2.CmdNext;
      S     #MotorUpSide2.CmdNext;
//--- Interlocking Motors
//RollsLowSide1
      A     #MDDx.Status.S1EnableMotors;
      ON    #Ma.Par.ParWithMDDx;
      A     #tmpEnable;
//[6.1]      U(    
//[6.1]      U     #HLOutlet1Side1.StFalse
//[6.1]      O     #HLOutlet1Side1.StCtoTrue
//[6.1]      ON    #Ma.Par.ParWithHLOutlet1Side1
//[6.1]      )     
//[6.1]      U(    
//[6.1]      U     #HLOutlet2Side1.StFalse
//[6.1]      O     #HLOutlet2Side1.StCtoTrue
//[6.1]      ON    #Ma.Par.ParWithHLOutlet2Side1
//[6.1]      )     
//[6.1]      U(                                //[6.0]
//[6.1]      U     #HLOutlet3Side1.StFalse     //[6.0]
//[6.1]      O     #HLOutlet3Side1.StCtoTrue   //[6.0]
//[6.1]      ON    #Ma.Par.ParWithHLOutlet3Side1    //[6.0]
//[6.1]      )                                 //[6.0]
      AN    #Ma.InDisableSide1;
      AN    #SM1Side1.StFault;
      AN    #MDDx.StFault;
      =     #MotorLowSide1.InEnableFwd;
// 
      A     #MDDx.OutComFault;	//[5.2]
      ON    #MDDx.Status.S1EnableMotors;	//[5.2]
      A     #Ma.Par.ParWithMDDx;	//[5.2]
      A(;	//[5.2]
      A     #MotorLowSide1.InManual;	//[5.2]
      O     #MotorUpSide1.InManual;	//[5.2]
      );	//[5.2]
      S     #MotorLowSide1.CmdOff;	//[5.2]
      S     #MotorUpSide1.CmdOff;	//[5.2]
// 
//RollsUpSide1
      A     #MotorLowSide1.StStartedFwd;
      AN    #Ma.InDisableSide1;
      A     #tmpEnable;
      =     #MotorUpSide1.InEnableFwd;
//SeqStop Side1
      A     #HLBackupLeftSide1.StFault;	//[6.0]
      A     #HLBackupLeftSide1.InpTrue;	//[6.0]
      O;	//[6.0]
      A     #HLBackupRightSide1.StFault;	//[6.0]
      A     #HLBackupRightSide1.InpTrue;	//[6.0]
      O     #tmpSeqStop;
      =     #MotorLowSide1.InSeqStop;
      =     #MotorUpSide1.InSeqStop;
//RollsLowSide2
      A     #MDDx.Status.S2EnableMotors;
      ON    #Ma.Par.ParWithMDDx;
      A     #tmpEnable;
//[6.1]      U(    
//[6.1]      U     #HLOutlet1Side2.StFalse
//[6.1]      O     #HLOutlet1Side2.StCtoTrue
//[6.1]      ON    #Ma.Par.ParWithHLOutlet1Side2
//[6.1]      )     
//[6.1]      U(    
//[6.1]      U     #HLOutlet2Side2.StFalse
//[6.1]      O     #HLOutlet2Side2.StCtoTrue
//[6.1]      ON    #Ma.Par.ParWithHLOutlet2Side2
//[6.1]      )     
//[6.1]      U(                                //[6.0]
//[6.1]      U     #HLOutlet3Side2.StFalse     //[6.0]
//[6.1]      O     #HLOutlet3Side2.StCtoTrue   //[6.0]
//[6.1]      ON    #Ma.Par.ParWithHLOutlet3Side2    //[6.0]
//[6.1]      )                                 //[6.0]
      AN    #Ma.InDisableSide2;
      AN    #SM1Side2.StFault;
      AN    #MDDx.StFault;
      =     #MotorLowSide2.InEnableFwd;
// 
      A     #MDDx.OutComFault;	//[5.2]
      ON    #MDDx.Status.S2EnableMotors;	//[5.2]
      A     #Ma.Par.ParWithMDDx;	//[5.2]
      A(;	//[5.2]
      A     #MotorLowSide2.InManual;	//[5.2]
      O     #MotorUpSide2.InManual;	//[5.2]
      );	//[5.2]
      S     #MotorLowSide2.CmdOff;	//[5.2]
      S     #MotorUpSide2.CmdOff;	//[5.2]
// 
//RollsUpSide2
      A     #MotorLowSide2.StStartedFwd;
      AN    #Ma.InDisableSide2;
      A     #tmpEnable;
      =     #MotorUpSide2.InEnableFwd;
//SeqStopSide2
      A     #HLBackupLeftSide2.StFault;	//[6.0]
      A     #HLBackupLeftSide2.InpTrue;	//[6.0]
      O;
      A     #HLBackupRightSide2.StFault;	//[6.0]
      A     #HLBackupRightSide2.InpTrue;	//[6.0]
      O;
      A     #tmpSeqStop;
      =     #MotorLowSide2.InSeqStop;
      =     #MotorUpSide2.InSeqStop;
NETWORK
TITLE = Interlockig MDDR/R
      A     #MotorUpSide1.StStartedFwd;
      O     #Ma.Par.Par4Rolls;
      ON    #Ma.Par.ParWithMotorUpSide1;	//[5.1]
      A     #MotorLowSide1.StStartedFwd;
      AN    #Ma.InDisableSide1;
      A     #Ma.InEnableDosing;
      =     #MDDx.Side1.InEnableDosing;
      A     #MotorUpSide2.StStartedFwd;
      O     #Ma.Par.Par4Rolls;
      ON    #Ma.Par.ParWithMotorUpSide2;	//[5.1]
      A     #MotorLowSide2.StStartedFwd;
      AN    #Ma.InDisableSide2;
      A     #Ma.InEnableDosing;
      =     #MDDx.Side2.InEnableDosing;
      A     #Ma.InOverrideHL;
      =     #MDDx.InOverrideHL;
//  RestDischarge
      A     #Ma.InRestDischarge;
      =     #MDDx.Side1.InRestdischarge;
      =     #MDDx.Side2.InRestdischarge;
NETWORK
TITLE = Help Signal
      NOP   0;
//Startup done
      A     #MotorLowSide1.StStartedFwd;
      A(;
      A     #MotorUpSide1.StStartedFwd;
      O     #MotorUpSide1.StFault;
      O     #Ma.Par.Par4Rolls;
      ON    #Ma.Par.ParWithMotorUpSide1;
      );
      O     #MotorLowSide1.StFault;	//[6.1]
      O     #Ma.InDisableSide1;
      A(;
      A     #MotorLowSide2.StStartedFwd;
      A(;
      O     #MotorUpSide2.StStartedFwd;
      O     #MotorUpSide2.StFault;
      O     #Ma.Par.Par4Rolls;
      ON    #Ma.Par.ParWithMotorUpSide2;
      );
      O     #MotorLowSide2.StFault;	//[6.1]
      O     #Ma.InDisableSide2;
      );
      =     #Ma.OutStartupDone;
//tmpStarted
      A     #MotorUpSide1.StStartedFwd;
      O     #Ma.Par.Par4Rolls;
      ON    #Ma.Par.ParWithMotorUpSide1;
      A     #MotorLowSide1.StStartedFwd;
      O     #Ma.InDisableSide1;
      A(;
      A     #MotorUpSide2.StStartedFwd;
      O     #Ma.Par.Par4Rolls;	//[3.2]
      ON    #Ma.Par.ParWithMotorUpSide2;
      A     #MotorLowSide2.StStartedFwd;
      O     #Ma.InDisableSide2;
      );
      A(;
      ON    #Ma.InDisableSide1;
      ON    #Ma.InDisableSide2;
      );
      =     #tmpStarted;
NETWORK
TITLE = Signal and DI from MDDX
      AN    #Ma.Par.ParWithMDDx;
      JC    MDJ1;
//--HLInlet---
      AN    #MDDx.Status.InpDI_0_4;
      =     #HLInletSide1.InpTrue;
      AN    #MDDx.Status.InpDI_0_16;
      =     #HLInletSide2.InpTrue;
      AN    #MDDx.Side1Divide.Out.OutHLInlet;
      =     #HLInletSide1Div.InpTrue;
      AN    #MDDx.Side1Divide.Out.OutHLInlet;
      =     #HLInletSide2Div.InpTrue;
//--HLBackup---
      AN    #MDDx.Side1.Out.OutStatus.OutHLBackupLeft;
      =     #HLBackupLeftSide1.InpTrue;
      AN    #MDDx.Side2.Out.OutStatus.OutHLBackupLeft;
      =     #HLBackupLeftSide2.InpTrue;
      AN    #MDDx.Side1.Out.OutStatus.OutHLBackupRight;
      =     #HLBackupRightSide1.InpTrue;
      AN    #MDDx.Side2.Out.OutStatus.OutHLBackupRight;
      =     #HLBackupRightSide2.InpTrue;
//--Motor---
      A     #MDDx.Side1.Out.OutLCAlarm.A055MotLow;
      =     #MotorLowSide1.InpFaultDev;
      A     #MDDx.Side1.Out.OutLCAlarm.A054MotUp;
      =     #MotorUpSide1.InpFaultDev;
      A     #MDDx.Side2.Out.OutLCAlarm.A055MotLow;
      =     #MotorLowSide2.InpFaultDev;
      A     #MDDx.Side2.Out.OutLCAlarm.A054MotUp;
      =     #MotorUpSide2.InpFaultDev;
//--HLOutlet
      AN    #MDDx.Status.InpDI_0_5;
      =     #HLOutlet1Side1.InpTrue;
      AN    #MDDx.Status.InpDI_0_6;
      =     #HLOutlet2Side1.InpTrue;
      AN    #MDDx.Status.InpDI_0_7;	//[6.0]
      =     #HLOutlet3Side1.InpTrue;	//[6.0]
      AN    #MDDx.Status.InpDI_0_17;
      =     #HLOutlet1Side2.InpTrue;
      AN    #MDDx.Status.InpDI_0_18;
      =     #HLOutlet2Side2.InpTrue;
      AN    #MDDx.Status.InpDI_0_19;	//[6.0]
      =     #HLOutlet3Side2.InpTrue;	//[6.0]
//--FU---
      L     #MDDx.Side1.Out.OutFeedRollSpeed;
      T     #FeedrollSide1.InOutValueUnits;
      L     0;
      >D;
      AN    #MDDx.StFault;
      A     #MDDx.Side1.InEnableDosing;
      NOT;
      =     #FeedrollSide1.InDisable;
      L     #MDDx.Side2.Out.OutFeedRollSpeed;
      T     #FeedrollSide2.InOutValueUnits;
      L     0;
      >D;
      AN    #MDDx.StFault;
      A     #MDDx.Side2.InEnableDosing;
      NOT;
      =     #FeedrollSide2.InDisable;
      L     #MDDx.Side1Divide.Out.OutFeedRollSpeed;
      T     #FeedrollSide1Div.InOutValueUnits;
      L     0;
      >D;
      AN    #MDDx.StFault;
      A     #MDDx.Side1.InEnableDosing;
      NOT;
      =     #FeedrollSide1Div.InDisable;
      L     #MDDx.Side2Divide.Out.OutFeedRollSpeed;
      T     #FeedrollSide2Div.InOutValueUnits;
      L     0;
      >D;
      AN    #MDDx.StFault;
      A     #MDDx.Side2.InEnableDosing;
      NOT;
      =     #FeedrollSide2Div.InDisable;
MDJ1: NOP   0;
NETWORK
TITLE = Call MotorLow
      CALL  #MotorLowSide1;
      CALL  #MotorLowSide2;
NETWORK
TITLE = Call Digital Input: SM Side1
      AN    #Ma.Par.ParWithSMSide1;
      JC    elL7;
      CALL  #SM1Side1;
elL7: NOP   0;
NETWORK
TITLE = Call Digital Input: SM1Side2
      AN    #Ma.Par.ParWithSMSide2;
      JC    elR6;
      CALL  #SM1Side2;
elR6: NOP   0;
NETWORK
TITLE = Call Digital Input: HLInletSide1
      AN    #Ma.Par.ParWithHLInletSide1;
      JC    elL5;
      CALL  #HLInletSide1;
elL5: NOP   0;
NETWORK
TITLE = Call Digital Input: HLInletSide2
      AN    #Ma.Par.ParWithHLInletSide2;
      JC    elR5;
      CALL  #HLInletSide2;
elR5: NOP   0;
NETWORK
TITLE = Call Digital Input: HLInletSide1Div
      AN    #Ma.Par.ParWithHLInletSide1Div;
      JC    elD1;
      CALL  #HLInletSide1Div;
elD1: NOP   0;
NETWORK
TITLE = Call Digital Input: HLInletSide1Div
      AN    #Ma.Par.ParWithHLInletSide2Div;
      JC    elD2;
      CALL  #HLInletSide2Div;
elD2: NOP   0;
NETWORK
TITLE = Call Digital Input: HLBackup
      A     #Ma.Par.Par4Rolls;
      JC    elL4;
      CALL  #HLBackupLeftSide1;
      CALL  #HLBackupRightSide1;
      CALL  #HLBackupLeftSide2;
      CALL  #HLBackupRightSide2;
elL4: NOP   0;
NETWORK
TITLE = Call MotorUpSide1
      A     #Ma.Par.Par4Rolls;
      ON    #Ma.Par.ParWithMotorUpSide1;
      JC    elL3;
      CALL  #MotorUpSide1;
elL3: NOP   0;
NETWORK
TITLE = Call MotorUpSide2
      A     #Ma.Par.Par4Rolls;
      ON    #Ma.Par.ParWithMotorUpSide2;
      JC    elR3;
      CALL  #MotorUpSide2;
elR3: NOP   0;
NETWORK
TITLE = Call MDDR
      AN    #Ma.Par.ParWithMDDx;
      JC    elMD;
      CALL  #MDDx;
elMD: NOP   0;
NETWORK
TITLE = Call Feedroll
      AN    #Ma.Par.ParWithMDDx;
      JC    elF9;
      CALL  #FeedrollSide1;
      CALL  #FeedrollSide2;
      AN    #MDDx.Par.ParSide1Divided;
      JC    elF4;
      CALL  #FeedrollSide1Div;
elF4: AN    #MDDx.Par.ParSide2Divided;
      JC    elF9;
      CALL  #FeedrollSide2Div;
elF9: NOP   0;
NETWORK
TITLE = Call Digital Input: HLOutlet
      AN    #Ma.Par.ParWithHLOutlet1Side1;
      JC    elO1;
      CALL  #HLOutlet1Side1;
elO1: AN    #Ma.Par.ParWithHLOutlet2Side1;
      JC    elO2;
      CALL  #HLOutlet2Side1;
elO2: AN    #Ma.Par.ParWithHLOutlet1Side2;
      JC    elO3;
      CALL  #HLOutlet1Side2;
elO3: AN    #Ma.Par.ParWithHLOutlet2Side2;
      JC    elO4;
      CALL  #HLOutlet2Side2;
elO4: AN    #Ma.Par.ParWithHLOutlet3Side1;
      JC    elH5;
      CALL  #HLOutlet3Side1;
elH5: AN    #Ma.Par.ParWithHLOutlet3Side2;
      JC    elH6;
      CALL  #HLOutlet3Side2;
elH6: NOP   0;
NETWORK
TITLE = Actual State
// StFault
      A     #tmpFaultSum;
      =     #Ma.StFault;
// StStopped
      A     #MotorUpSide1.StStopped;
      O     #Ma.Par.Par4Rolls;
      ON    #Ma.Par.ParWithMotorUpSide1;	//[5.1]
      A(;
      A     #MotorUpSide2.StStopped;
      O     #Ma.Par.Par4Rolls;
      ON    #Ma.Par.ParWithMotorUpSide2;	//[5.1]
      );
      A     #MotorLowSide1.StStopped;
      A     #MotorLowSide2.StStopped;
      AN    #Ma.StFault;
      =     #Ma.StStopped;
// StEngaged
      A     #MDDx.Side1.StEngaged;
      O     #MDDx.Side2.StEngaged;
      A     #tmpStarted;
      AN    #Ma.StFault;
      AN    #Ma.StStopped;
      =     #Ma.StEngaged;
// StStarted
      A     #tmpStarted;
      AN    #Ma.StFault;
      AN    #Ma.StStopped;
      AN    #Ma.StEngaged;
      =     #Ma.StStarted;
// StStopping
      A     #MotorLowSide1.InSeqStop;
      O     #MotorLowSide2.InSeqStop;
      AN    #Ma.StStarted;
      AN    #Ma.StStopped;
      AN    #Ma.StFault;
      AN    #Ma.StEngaged;
      =     #Ma.StStopping;
// StStarting
      AN    #Ma.StStopped;
      AN    #Ma.StStarted;
      AN    #Ma.StStopping;
      AN    #Ma.StFault;
      AN    #Ma.StEngaged;
      =     #Ma.StStarting;
NETWORK
TITLE = State Code
// State     StCode
// ----------------------
// StFault32
// StStopped    1
// StStarting   2
// StStarted   3
// StEngaged   4 
// StStopping  7
      A     #Ma.StStopped;
      L     1;	//Code=StStopped
      JC    Code;
      A     #Ma.StStarted;
      L     3;	//Code=StStarted
      JC    Code;
      A     #Ma.StEngaged;
      L     4;	//Code=StEngaged
      JC    Code;
      A     #Ma.StStarting;
      L     2;	//Code=StStarting
      JC    Code;
      A     #Ma.StStopping;
      L     7;	//Code=StStopping 
      JC    Code;
      L     32;	//Code=StFault 
//----------------------
Code: L     #Ma.StCode;	// Old state code
      TAK;
      T     #Ma.StCode;	// Save state code
      <>I;
      L     3;
      CC    "SYS_CBitCtrl";	//Set change bit
NETWORK
TITLE = Global End
      NOP   0;
//---Clear all commands
      CLR;
      =     #Ma.CmdOn;
      =     #Ma.CmdOff;
      =     #Ma.CmdNext;
      =     #Ma.CmdFaultReset;
//Monitoring / Prealarm
//  --HL Inlet
      A     #HLInletSide1.InpTrue;	//[6.0]
      AN    #Ma.InOverrideHL;
      =     #HLInletSide1.InMonFalse;
      A     #HLInletSide2.InpTrue;	//[6.0]
      AN    #Ma.InOverrideHL;
      =     #HLInletSide2.InMonFalse;
      A     #HLInletSide1Div.InpTrue;	//[6.0]
      AN    #Ma.InOverrideHL;
      =     #HLInletSide1Div.InMonFalse;
      A     #HLInletSide2Div.InpTrue;	//[6.0]
      AN    #Ma.InOverrideHL;
      =     #HLInletSide2Div.InMonFalse;
END_FUNCTION_BLOCK

FUNCTION_BLOCK "GCS7_Ma_DischagerFlat"	// FB 88
TITLE = Bin discharger A
//COPYRIGHT:    (C) 1997  BUHLER AG, CH-9240 UZWIL, SWITZERLAND
//
//PRODUCT:      GCS7
//
//TITLE:        FB 88 Machine Bin discharger Flat-Bottom
//
//-------------------------------------------------------------------------
//
//IDENT:        AUTHOR:             DEPT:                       DATE:
//
//FB88.1.1      A. Egli             BASE                        02-Mar-2009
//              Update J.Chische
//FB88.1.0      A. Egli             BASE                        24-Jul-2008
//              1st Release in S7
//
//-------------------------------------------------------------------------
//
//PURPOSE:      MANUAL : see [LL.DSAxxMAN]
//
//RESTRICTIONS: S7
//
//-------------------------------------------------------------------------
//
//
AUTHOR : EA
FAMILY : GCS7LL
NAME : Discharg
VERSION : 1.1
VAR
  Ma : UDT 20880;
  Discharger : FB 13;	//Element
  LL : FB 14;	//Element
  Sweeper : FB 12;	//Element (de: Räumer)
  SwitchSweeper : FB 14;	//Element (de: Schalter Start räumen)
  Slide1 : FB 13;	//Element (de: Seitlicher Auslaufschieber 1)
  Slide2 : FB 13;	//Element (de: Seitlicher Auslaufschieber 2)
  Slide3 : FB 13;	//Element (de: Seitlicher Auslaufschieber 3)
  Slide4 : FB 13;	//Element (de: Seitlicher Auslaufschieber 4)
END_VAR
VAR_TEMP
  tmpFaultStop : BOOL ;
  tmpFaultSum : BOOL ;
  tmpNext : BOOL ;
  tmpLenDyn : INT ;
  tmpStoreAR2 : DINT ;
END_VAR
BEGIN
NETWORK
TITLE =
      L     20;
      T     #tmpLenDyn;
NETWORK
TITLE = PC Control
//=== Test Object number =====================
      L     "SYS_DirectCtrlDB".PC.ObjectNo;	//PCControl.ObjectNo
      L     #Ma.Par.ParObjectNo;	//Input ObjectNo
      <>I;
      JC    aEnd;
//=== Test OType      ========================
      L     2088;	//Input object type
      L     "SYS_DirectCtrlDB".PC.ObjectType;	//PCControl.ObjectType
      <>I;
      JC    aEnd;
//=== Test Handshake =========================
      A     "SYS_DirectCtrlDB".PC.Hsk.FExamine;	// Handshake.FExamine
      JC    aExa;
      A     "SYS_DirectCtrlDB".PC.Hsk.FDefineCmd;	// Handshake.FDefineCmd
      JC    aCmd;
      A     "SYS_DirectCtrlDB".PC.Hsk.FDefinePara;	// Handshake.FDefinePara
      JC    aPar;
aIni: L     2;	// FcInit
      UC    "SYS_DirectCtrl";
      JU    aEnd;
// Write parameter 
aPar: LAR1  P#DBX 58.0;
      L     P#6.0;
      +AR1;
// Write new commands from PC to Interface of group 
aCmd: A     "SYS_DirectCtrlDB".PC.Cmd1[8];	//Cmd1[8]=CmdOff
      S     #Ma.CmdOff;
      A     "SYS_DirectCtrlDB".PC.Cmd1[9];	//Cmd1[9]=CmdOn
      S     #Ma.CmdOn;
      A     "SYS_DirectCtrlDB".PC.Cmd1[10];	//Cmd1[10]=CmdNext
      S     #Ma.CmdNext;
      A     "SYS_DirectCtrlDB".PC.Cmd1[11];	//Cmd1[11]=CmdFaultReset
      S     #Ma.CmdFaultReset;
      A     "SYS_DirectCtrlDB".PC.Cmd1[13];	//Cmd1[13]=CmdManualOn
      S     #Ma.InManual;
      A     "SYS_DirectCtrlDB".PC.Cmd1[1];	//Cmd1[1]=CmdRestDischargeOn
      S     #Ma.InRestDischarge;
      A     "SYS_DirectCtrlDB".PC.Cmd2[1];	//Cmd2[1]=CmdRestDischargeOff
      R     #Ma.InRestDischarge;
      JU    aIni;
aExa: TAR2;	// Address Dynamic data
      T     "SYS_DirectCtrlDB".GC.InDynAddr;	// -->PCControl.GC.InDynAddr
      L     #tmpLenDyn;	// Length Dynamic data
      T     "SYS_DirectCtrlDB".GC.InDynLen;	// -->PCControl.GC.InDynLen
      L     0;
      T     "SYS_DirectCtrlDB".GC.InParaAddr;	// -->PCControl.GC.InParaAddr
      T     "SYS_DirectCtrlDB".GC.InParaLen;	// -->PCControl.GC.InParaLen
      L     1;	// Code FcExamine
      UC    "SYS_DirectCtrl";
      L     10;	//Revision
      T     "SYS_DirectCtrlDB".GC.Revision;
aEnd: NOP   0;
NETWORK
TITLE = Interlocking
//===Global Group Orders===
      A     "GCS7_Gr_OutManualOn";	//Gr.OutManualOn
      S     #Ma.InManual;
      A     "GCS7_Gr_OutManualOff";	//Gr.OutManualOff
      R     #Ma.InManual;
      A     #Ma.InManual;
      S     "GCS7_Gr_InManual";	//Gr.InManual
      A     #Ma.CmdNext;
      AN    #Ma.InManual;
      O     #Ma.CmdOn;
      =     #tmpNext;
//---- Low level 
//--- Fault----
      A     #Discharger.StFault;
      O     #LL.StFault;
      O     #Sweeper.StFault;
      O     #SwitchSweeper.StFault;
      O     #Slide1.StFault;
      O     #Slide2.StFault;
      O     #Slide3.StFault;
      O     #Slide4.StFault;
      =     #tmpFaultSum;
// 
//--- Local mode --
      A     #Ma.InLocal;
      AN    #Ma.InManual;
      =     #Discharger.InLocal;
      =     #LL.InLocal;
      =     #Sweeper.InLocal;
      =     #SwitchSweeper.InLocal;
      CLR;
      =     #Slide1.InLocal;
      =     #Slide2.InLocal;
      =     #Slide3.InLocal;
      =     #Slide4.InLocal;
//--- Fault Reset -------------
      A     #Ma.CmdFaultReset;
      S     #Discharger.CmdFaultReset;
      S     #LL.CmdFaultReset;
      S     #Sweeper.CmdFaultReset;
      S     #SwitchSweeper.CmdFaultReset;
      S     #Slide1.CmdFaultReset;
      S     #Slide2.CmdFaultReset;
      S     #Slide3.CmdFaultReset;
      S     #Slide4.CmdFaultReset;
//--- Interlocking Discharger 
      A     #Ma.InEnable;
      A     #tmpNext;
      S     #Discharger.InEnableHN;	//Discharger.InEnableHN; 
      S     #Discharger.CmdNext;
      AN    #Ma.InEnable;
      O     #Ma.CmdOff;
      R     #Discharger.InEnableHN;	//Discharger.InEnableHN; 
      AN    #Discharger.InEnableHN;
      =     #Discharger.InEnableLN;
      S     #Discharger.CmdNext;
//--- Interlocking SwitchSweeper 
      AN    #Ma.InRestDischarge;
      =     #SwitchSweeper.InMonFalse;
//--- Interlocking Sweeper 
      A(;	//-jc- [1.1]
      A     #Slide1.StHN;	//-jc- [1.1] 
      ON    #Ma.Par.ParWithSlide1;	//-jc- [1.1]
      );	//-jc- [1.1]
      O(;	//-jc- [1.1]
      A     #Slide2.StHN;	//-jc- [1.1]
      ON    #Ma.Par.ParWithSlide2;	//-jc- [1.1]
      );	//-jc- [1.1]
      O(;	//-jc- [1.1]
      A     #Slide3.StHN;	//-jc- [1.1]
      ON    #Ma.Par.ParWithSlide3;	//-jc- [1.1]
      );	//-jc- [1.1]
      O(;	//-jc- [1.1]
      A     #Slide4.StHN;	//-jc- [1.1]
      ON    #Ma.Par.ParWithSlide4;	//-jc- [1.1]
      );	//-jc- [1.1]
//      U     #LL.StFalse                 //Unvovered---jc- [1.1]
      A     #Discharger.StHN;
      A     #Ma.InEnable;
      A     #SwitchSweeper.InpTrue;
      A     #Ma.InDoorOpen;
      A     #Ma.InRestDischarge;
      =     #Sweeper.InEnableFwd;
      A     #Sweeper.InEnableFwd;
      A     #LL.StFalse;	//-jc- [1.1]
      S     #Sweeper.CmdNext;
//--- Interlocking Slide 
      AN    #LL.StFalse;	//Unvovered
      AN    #Ma.InDoorOpen;	//-jc- [1.1]
      ON    #Ma.InRestDischarge;
//      ON    #Discharger.StHN          //-jc- [1.1]
      =     #Slide1.InEnableLN;
      =     #Slide2.InEnableLN;
      =     #Slide3.InEnableLN;
      =     #Slide4.InEnableLN;
      SET;
      S     #Slide1.CmdNext;
      S     #Slide2.CmdNext;
      S     #Slide3.CmdNext;
      S     #Slide4.CmdNext;
//--- Interlocking discharge conveying 
      A(;
      A     #Slide1.StLN;
      ON    #Ma.Par.ParWithSlide1;
      );
      A(;
      A     #Slide2.StLN;
      ON    #Ma.Par.ParWithSlide2;
      );
      A(;
      A     #Slide3.StLN;
      ON    #Ma.Par.ParWithSlide3;
      );
      A(;
      A     #Slide4.StLN;
      ON    #Ma.Par.ParWithSlide4;
      );
      O     #Ma.InRestDischarge;	//-jc- [1.1]
      AN    #Slide1.StFault;
      AN    #Slide2.StFault;
      AN    #Slide3.StFault;
      AN    #Slide4.StFault;
      =     #Ma.OutEnableConveying;
NETWORK
TITLE = Call Discharger
      CALL  #Discharger;
NETWORK
TITLE = Call LL
      CALL  #LL;
NETWORK
TITLE = Call Sweep
      CALL  #Sweeper;
NETWORK
TITLE = Call SwitchSweep
      CALL  #SwitchSweeper;
NETWORK
TITLE = Call Slide1
      AN    #Ma.Par.ParWithSlide1;
      JC    ELS1;
      CALL  #Slide1;
ELS1: NOP   0;
NETWORK
TITLE = Call Slide2
      AN    #Ma.Par.ParWithSlide2;
      JC    ELS2;
      CALL  #Slide2;
ELS2: NOP   0;
NETWORK
TITLE = Call Slide3
      AN    #Ma.Par.ParWithSlide3;
      JC    ELS3;
      CALL  #Slide3;
ELS3: NOP   0;
NETWORK
TITLE = Call Slide4
      AN    #Ma.Par.ParWithSlide4;
      JC    ELS4;
      CALL  #Slide4;
ELS4: NOP   0;
NETWORK
TITLE = Jump to actual state
      A     #Ma.StStopped;
      JC    S0;	// ===> State
      A     #Ma.StStarted;
      JC    S2;	// ===> State
      A     #Ma.StStarting;
      JC    S1;	// ===> State
      A     #Ma.StStopping;
      JC    S3;	// ===> State
      A     #Ma.StFault;
      JC    S4;	// ===> State
NETWORK
TITLE = Stopped
//any Transition 
xxS0: S     #Ma.StStopped;	// ===> Initialisation
      JU    OUT;
//=== Logic
// Condition for StFault
S0:   A     #tmpFaultSum;
      R     #Ma.StStopped;
      JC    xxS4;	//--> ST_FAULT:
// Condition for StStarting
      AN    #Discharger.StLN;
      R     #Ma.StStopped;
      JC    xxS1;	//--> StStarting
      JU    OUT;
NETWORK
TITLE = StStarting
//any Transition 
xxS1: S     #Ma.StStarting;
      JU    OUT;
//=== Logic
// Condition for StFault
S1:   A     #tmpFaultSum;
      R     #Ma.StStarting;
      JC    xxS4;	//--> StFault
// Condition for StStarted
      A     #Discharger.StHN;
      R     #Ma.StStarting;
      JC    xxS2;	//-->StStarted
// Condition for StStopping
      AN    #Discharger.StCtoHN;
      R     #Ma.StStarting;
      JC    xxS3;	//-->StStopping
      JU    OUT;
NETWORK
TITLE = StStarted
//any Transition 
xxS2: S     #Ma.StStarted;
      JU    OUT;
//=== Logic
// Condition for StFault
S2:   A     #tmpFaultSum;
      R     #Ma.StStarted;
      JC    xxS4;	//--> StFault
// Condition for StStopping
      AN    #Discharger.StHN;
      R     #Ma.StStarted;
      JC    xxS3;	//-->StStopping
      JU    OUT;
NETWORK
TITLE = Stopping
//any Transition 
xxS3: S     #Ma.StStopping;
      JU    OUT;
//=== Logic
// Condition for StFault
S3:   A     #tmpFaultSum;
      R     #Ma.StStopping;
      JC    xxS4;	//--> StFault
// Condition for StStopped
      A     #Discharger.StLN;
      R     #Ma.StStopping;
      JC    xxS0;	//-->StStopped
// Condition for StStarting
      AN    #Discharger.StCtoLN;
      AN    #Discharger.StLN;
      R     #Ma.StStopping;
      JC    xxS1;	//-->StStarting
      JU    OUT;
NETWORK
TITLE = Fault
//any Transition 
xxS4: S     #Ma.StFault;
      JU    OUT;
//=== Logic
S4:   A     #tmpFaultSum;
      JC    OUT;
//---- Transition --
      R     #Ma.StFault;
      JU    xxS0;	//-->StStopping 
NETWORK
TITLE = State Code
// State     StCode
// ----------------------
// StFault32
// StStopped       1
// StStarting      2
// StStarted       3
// StStopping      7
// StRestDischarge 9
//
OUT:  A     #Ma.StStopped;
      L     1;	//Code=StStopped
      JC    Code;
      L     9;	//Code: emptying
      A     #LL.StFalse;
      A     #Ma.InRestDischarge;
      A     #Ma.StStarted;
      JC    Code;
      A     #Ma.StStarted;
      L     3;	//Code=StStarted
      JC    Code;
      A     #Ma.StStarting;
      L     2;	//Code=StStarting
      JC    Code;
      A     #Ma.StStopping;
      L     7;	//Code=StStopping 
      JC    Code;
      L     32;	//Code=StFault 
Code: L     #Ma.StCode;	// Old state code
      TAK;
      T     #Ma.StCode;	// Save state code
      <>I;
      L     3;
      CC    "SYS_CBitCtrl";	//Set change bit
NETWORK
TITLE = Global End
      CLR;	//---Clear all commands
      =     #Ma.CmdOn;
      =     #Ma.CmdOff;
      =     #Ma.CmdNext;
      =     #Ma.CmdFaultReset;
END_FUNCTION_BLOCK

